REGION Network 2: kontrola przebiegu pętli odczytu parametró z modbus rtu
   RUNG wire#powerrail
      Contact( "dbTags_master_MPP04_2".modbusMaster.busy )
      { S7_Templates := "time_type := Time" } "IEC_Timer_loop_rtu_error_DB".TON(pt := "dbTimersForDrivers".error_loop_modbus_rtu.PT, et =>)
      Coil( "comunication_alarm_modbus_rtu" )
   END_RUNG
   // the same network as SCL:
   "IEC_Timer_loop_rtu_error_DB".TON(IN := "dbTags_master_MPP04_2".modbusMaster.busy,
                           PT := "dbTimersForDrivers".error_loop_modbus_rtu.PT);
   "comunication_alarm_modbus_rtu" := "IEC_Timer_loop_rtu_error_DB".Q;
END_REGION

REGION Network 3: przekazanie do zmiennej error status
   // jeśli wystąpił błąd to przenieś 8200 ( kod brak urządzenia na linni)
   RUNG wire#powerrail
      I_Contact( "FirstScan" )
      Contact( "comunication_alarm_modbus_rtu" )
      Move(in := 33280, out1 => "dbTags_master_MPP04_2".modbusMaster.errorStatus)
   END_RUNG
   // the same network as SCL:
   IF NOT "FirstScan" AND "comunication_alarm_modbus_rtu" THEN
       "dbTags_master_MPP04_2".modbusMaster.errorStatus := 33280;
   END_IF;
END_REGION
END_FUNCTION_BLOCK

ORGANIZATION_BLOCK "Cyclic interrupt"   // OB31, LAD, CyclicInterrupt
{ S7_Optimized_Access := 'TRUE' }
VERSION : 0.1
// stored: AutoNumber true, IsIECCheckEnabled false, SetENOAutomatically false
   VAR_INPUT
      Initial_Call : Bool;   // Initial call of this OB
      Event_Count : Int;   // Events discarded
   END_VAR
   VAR_TEMP
      disconect : Bool;
   END_VAR
BEGIN

REGION Network 1: Reset znacznika automatycznego przekazania wartości na zamykanie
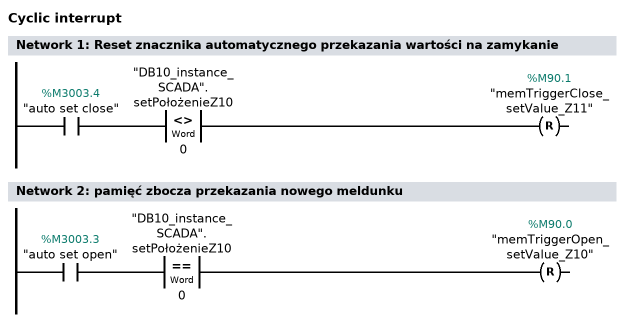
   RUNG wire#powerrail
      Contact( "auto set close" )
      { S7_Templates := "SrcType := Word" } NE_Contact(in1 := "DB10_instance_SCADA".setPołożenieZ10, in2 := 0)
      R_Coil( "memTriggerClose_setValue_Z11" )
   END_RUNG
   // the same network as SCL:
   IF "auto set close" AND ("DB10_instance_SCADA".setPołożenieZ10 <> 0) THEN
       "memTriggerClose_setValue_Z11" := FALSE;
   END_IF;
END_REGION

REGION Network 2: pamięć zbocza przekazania nowego meldunku
   RUNG wire#powerrail
      Contact( "auto set open" )
      { S7_Templates := "SrcType := Word" } EQ_Contact(in1 := "DB10_instance_SCADA".setPołożenieZ10, in2 := 0)
      R_Coil( "memTriggerOpen_setValue_Z10" )
   END_RUNG
   // the same network as SCL:
   IF "auto set open" AND ("DB10_instance_SCADA".setPołożenieZ10 = 0) THEN
       "memTriggerOpen_setValue_Z10" := FALSE;
   END_IF;
END_REGION

REGION Network 3 (SCL): Reset znaczników zbocza wysyłania danych przez TCP
   "memRisingTriger_Data_1" := FALSE;
   "memTrig_Client_Receiving_1" := FALSE;
   "memRisingTriger_Data_2" := FALSE;
   "memTrig_Client_Receiving_2" := FALSE;
   "memRisingTriger_Data_3" := FALSE;
   "memTrig_Client_Receiving_3" := FALSE;
   "memRisingTriger_Data_4" := FALSE;
   "memTrig_Client_Receiving_4" := FALSE;
   "memRisingTriger_Data_5" := FALSE;
   "memTrig_Client_Receiving_5" := FALSE;
   "memRisingTriger_Data_6" := FALSE;
   "memTrig_Client_Receiving_6" := FALSE;
   "memRisingTriger_Data_7" := FALSE;
   "memTrig_Client_Receiving_7" := FALSE;
   "memRisingTriger_Data_8" := FALSE;
   "memTrig_Client_Receiving_8" := FALSE;
   "memRisingTriger_Data_9" := FALSE;
   "memTrig_Client_Receiving_9" := FALSE;
   "memRisingTriger_Data_10" := FALSE;
   "memTrig_Client_Receiving_10" := FALSE;
END_REGION

REGION Network 4 (SCL): pamieć zbocza zmiany danych w zmiennej
   "memRisingTriger_Data_11" := FALSE;
   "memTrig_Client_Receiving_11" := FALSE;
   "memRisingTriger_Data_12" := FALSE;
   "memTrig_Client_Receiving_12" := FALSE;
   "memRisingTriger_Data_13" := FALSE;
   "memTrig_Client_Receiving_13" := FALSE;
   "memRisingTriger_Data_14" := FALSE;
   "memTrig_Client_Receiving_14" := FALSE;
   "memRisingTriger_Data_15" := FALSE;
   "memTrig_Client_Receiving_15" := FALSE;
   "memRisingTriger_Data_16" := FALSE;
   "memTrig_Client_Receiving_16" := FALSE;
   "memRisingTriger_Data_17" := FALSE;
   "memTrig_Client_Receiving_17" := FALSE;
   "memRisingTriger_Data_18" := FALSE;
   "memTrig_Client_Receiving_18" := FALSE;
   "memRisingTriger_Data_19" := FALSE;
   "memTrig_Client_Receiving_19" := FALSE;
   "memRisingTriger_Data_20" := FALSE;
   "memTrig_Client_Receiving_20" := FALSE;
END_REGION

REGION Network 5: pamieć zbocza narastającego przekazania danej do wysłania
END_REGION
END_ORGANIZATION_BLOCK

ORGANIZATION_BLOCK "Cyclic interrupt_ModbusTCP_wysyłanie"   // OB30, LAD, CyclicInterrupt
{ S7_Optimized_Access := 'TRUE' }
VERSION : 0.1
// stored: AutoNumber true, IsIECCheckEnabled false, SetENOAutomatically false
   VAR_INPUT
      Initial_Call : Bool;   // Initial call of this OB
      Event_Count : Int;   // Events discarded
   END_VAR
BEGIN

REGION Network 1: Odczyt poziomów w zbiornku
END_REGION

REGION Network 2 (SCL): Odczyt poziomów w zbiornku
   "AI_poziom_zbiornik_1" := "IW68";
   "AI_poziom_zbiornik_2" := "IW70";
   "AI_poziom_zbiornik_3" := "IW72";
   "AI_poziom_zbiornik_4" := "IW74";

   "AI_położenie_Z10" := "IW78";
END_REGION

REGION Network 3 (SCL): Ciśnienie magistrala

   IF "IW76":P > 0.2 THEN // czy nie uszkodzone rury
     IF "IW76":P < 27651 THEN // przerwana pętla prądowa
       // to przekazanie wartości
       "AI_ciśnienie_B5" := "IW76":P;
       ;
     ELSE
       "AI_ciśnienie_B5" := 32767;
       ;
     END_IF;

     ;
   END_IF;
END_REGION

REGION Network 4 (SCL): Położenie zasuwy Z10
   // Odczyt w FC5
END_REGION
END_ORGANIZATION_BLOCK

ORGANIZATION_BLOCK "Cyclic interrupt_WatchDog_comunication"   // OB32, LAD, CyclicInterrupt
TITLE = Kontrola komunikacji TCP, HMI, PLC
{ S7_Optimized_Access := 'TRUE' }
AUTHOR : rtecmer
VERSION : 0.1
// stored: AutoNumber true, IsIECCheckEnabled false, SetENOAutomatically false
   VAR_INPUT
      Initial_Call : Bool;   // Initial call of this OB
      Event_Count : Int;   // Events discarded
   END_VAR
BEGIN

REGION Network 1
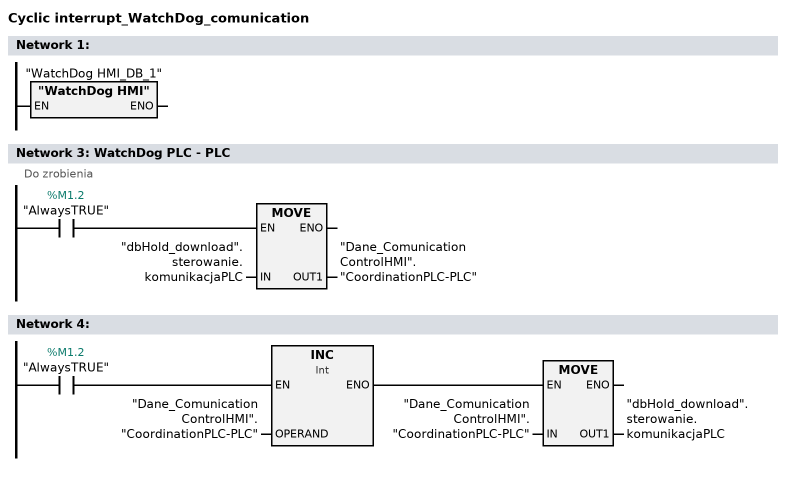
   RUNG wire#powerrail
      "WatchDog HMI_DB_1"()
   END_RUNG
   // the same network as SCL:
   "WatchDog HMI_DB_1"();   // "WatchDog HMI"
END_REGION

REGION Network 3: WatchDog PLC - PLC
   // Do zrobienia
   RUNG wire#powerrail
      Contact( "AlwaysTRUE" )
      Move(in := "dbHold_download".sterowanie.komunikacjaPLC, out1 => "Dane_ComunicationControlHMI"."CoordinationPLC-PLC")
   END_RUNG
   // the same network as SCL:
   IF "AlwaysTRUE" THEN
       "Dane_ComunicationControlHMI"."CoordinationPLC-PLC" := "dbHold_download".sterowanie.komunikacjaPLC;
   END_IF;
END_REGION

REGION Network 4
   RUNG wire#powerrail
      Contact( "AlwaysTRUE" )
      { S7_Templates := "DestType := Int" } Inc( "Dane_ComunicationControlHMI"."CoordinationPLC-PLC" )
      Move(in := "Dane_ComunicationControlHMI"."CoordinationPLC-PLC", out1 => "dbHold_download".sterowanie.komunikacjaPLC)
   END_RUNG
   // the same network as SCL:
   IF "AlwaysTRUE" THEN
       "Dane_ComunicationControlHMI"."CoordinationPLC-PLC" := "Dane_ComunicationControlHMI"."CoordinationPLC-PLC" + 1;
       "dbHold_download".sterowanie.komunikacjaPLC := "Dane_ComunicationControlHMI"."CoordinationPLC-PLC";
   END_IF;
END_REGION

REGION Network 6 (SCL): kasowanie znacznków HMI
   // znaczniki HMI do kasowania alrmów ekranów
   "dbtags_Sterowanie".HMI.resetScreen_1 := FALSE;
   "dbtags_Sterowanie".HMI.resetScreen_2 := FALSE;
   "dbtags_Sterowanie".HMI.resetScreen_3 := FALSE;
   "dbtags_Sterowanie".HMI.resetScreen_4 := FALSE;
   "dbtags_Sterowanie".HMI.resetScreen_5 := FALSE;
   "dbtags_Sterowanie".HMI.resetScreen_6 := FALSE;
   "dbtags_Sterowanie".HMI.resetScreen_7 := FALSE;
   "dbtags_Sterowanie".HMI.resetScreen_8 := FALSE;
END_REGION
END_ORGANIZATION_BLOCK

FUNCTION_BLOCK "WatchDog HMI"   // FB12, LAD
TITLE = WatchDog HMI
{ S7_Optimized_Access := 'TRUE' }
AUTHOR : rtecmer
VERSION : 0.1
// Kontrola komunikacji PLC z HMI. Informacja o zerwanym połączeniu przekazywana do DB SCADA WinCC
// stored: AutoNumber true, IsIECCheckEnabled false, IsRetainMemResEnabled false, MemoryReserve 500, SetENOAutomatically false, UDAEnableTagReadback false
   VAR_TEMP   // added for the SCL form of the ladder/FBD networks
      _w1 : Bool;
      _w2 : Bool;
   END_VAR
BEGIN

REGION Network 1: WatchDog HMI
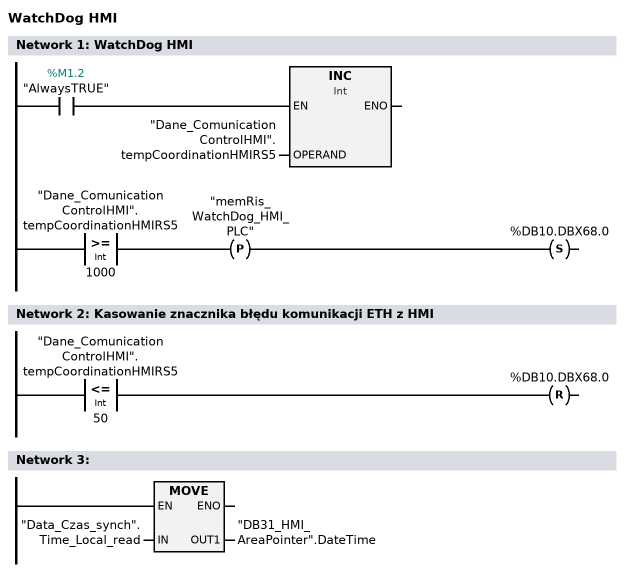
   RUNG wire#powerrail
      Contact( "AlwaysTRUE" )
      { S7_Templates := "DestType := Int" } Inc( "Dane_ComunicationControlHMI".tempCoordinationHMIRS5 )
   END_RUNG
   RUNG wire#powerrail
      { S7_Templates := "SrcType := Int" } GE_Contact(in1 := "Dane_ComunicationControlHMI".tempCoordinationHMIRS5, in2 := 1000)
      P_Trig( "memRis_WatchDog_HMI_PLC" )
      S_Coil( %DB10.DBX68.0 )
   END_RUNG
   // the same network as SCL:
   IF "AlwaysTRUE" THEN
       "Dane_ComunicationControlHMI".tempCoordinationHMIRS5 := "Dane_ComunicationControlHMI".tempCoordinationHMIRS5 + 1;
   END_IF;
   #_w1 := "Dane_ComunicationControlHMI".tempCoordinationHMIRS5 >= 1000;
   #_w2 := #_w1 AND NOT "memRis_WatchDog_HMI_PLC";   // rising edge
   "memRis_WatchDog_HMI_PLC" := #_w1;
   IF #_w2 THEN %DB10.DBX68.0 := TRUE; END_IF;
END_REGION

REGION Network 2: Kasowanie znacznika błędu komunikacji ETH z HMI
   RUNG wire#powerrail
      { S7_Templates := "SrcType := Int" } LE_Contact(in1 := "Dane_ComunicationControlHMI".tempCoordinationHMIRS5, in2 := 50)
      R_Coil( %DB10.DBX68.0 )
   END_RUNG
   // the same network as SCL:
   IF "Dane_ComunicationControlHMI".tempCoordinationHMIRS5 <= 50 THEN %DB10.DBX68.0 := FALSE; END_IF;
END_REGION

REGION Network 3
   RUNG wire#powerrail
      Move(in := "Data_Czas_synch".Time_Local_read, out1 => "DB31_HMI_AreaPointer".DateTime)
   END_RUNG
   // the same network as SCL:
   "DB31_HMI_AreaPointer".DateTime := "Data_Czas_synch".Time_Local_read;
END_REGION
END_FUNCTION_BLOCK

ORGANIZATION_BLOCK "Diagnostic error interrupt"   // OB82, LAD, DiagnosticErrorInterrupt
{ S7_Optimized_Access := 'TRUE' }
VERSION : 0.1
// stored: IsIECCheckEnabled false, SetENOAutomatically false
   VAR_INPUT
      IO_State : Word;   // IO state of the HW object
      LADDR : HW_ANY;   // Hardware identifier
      Channel : UInt;   // Channel number
      MultiError : Bool;   // =true if more than one error is present
   END_VAR
   VAR_TEMP
      RetVal_RD_SYS_T : Int;   // //Status of the instruction RD_SYS_T: Read time-of-day
   END_VAR
BEGIN

REGION Network 2 (SCL)
   "EX012_ErrorBuffer_OB82".OB82ErrorCounter := "EX012_ErrorBuffer_OB82".OB82ErrorCounter + 1;
   //ochrona przed przepełnieniem tabeli
   IF ("EX012_ErrorBuffer_OB82".OB82ErrorCounter > "CONST_BUFFER_OB82") THEN
     "EX012_ErrorBuffer_OB82".OB82ErrorCounter := 1;
   END_IF;
   //Wystąpił błąd czasu
   #RetVal_RD_SYS_T := RD_LOC_T(OUT => "EX012_ErrorBuffer_OB82".ErrorDataOB82["EX012_ErrorBuffer_OB82".OB82ErrorCounter].ErrorTimestamp);
   //Zapis błedu do buffora (ErrorBuffor)
   "EX012_ErrorBuffer_OB82".ErrorDataOB82["EX012_ErrorBuffer_OB82".OB82ErrorCounter].IO_State := #IO_State;
   "EX012_ErrorBuffer_OB82".ErrorDataOB82["EX012_ErrorBuffer_OB82".OB82ErrorCounter].LADDR := #LADDR;
   "EX012_ErrorBuffer_OB82".ErrorDataOB82["EX012_ErrorBuffer_OB82".OB82ErrorCounter].Channel := #Channel;
   "EX012_ErrorBuffer_OB82".ErrorDataOB82["EX012_ErrorBuffer_OB82".OB82ErrorCounter].MultiError := #MultiError;
END_REGION
END_ORGANIZATION_BLOCK

ORGANIZATION_BLOCK "Startup"   // OB100, LAD, Startup
TITLE = "Complete Restart"
{ S7_Optimized_Access := 'TRUE' }
VERSION : 0.1
// Zasuwa status aut. zamknięta= 35980
// Zasuwa status aut. otwarta=34438
// stored: AutoNumber true, IsIECCheckEnabled false, SetENOAutomatically false
   VAR_INPUT
      LostRetentive : Bool;   // True if retentive data are lost
      LostRTC : Bool;   // True if date and time are lost
   END_VAR
BEGIN

REGION Network 1: znacznik powrotu zasilania
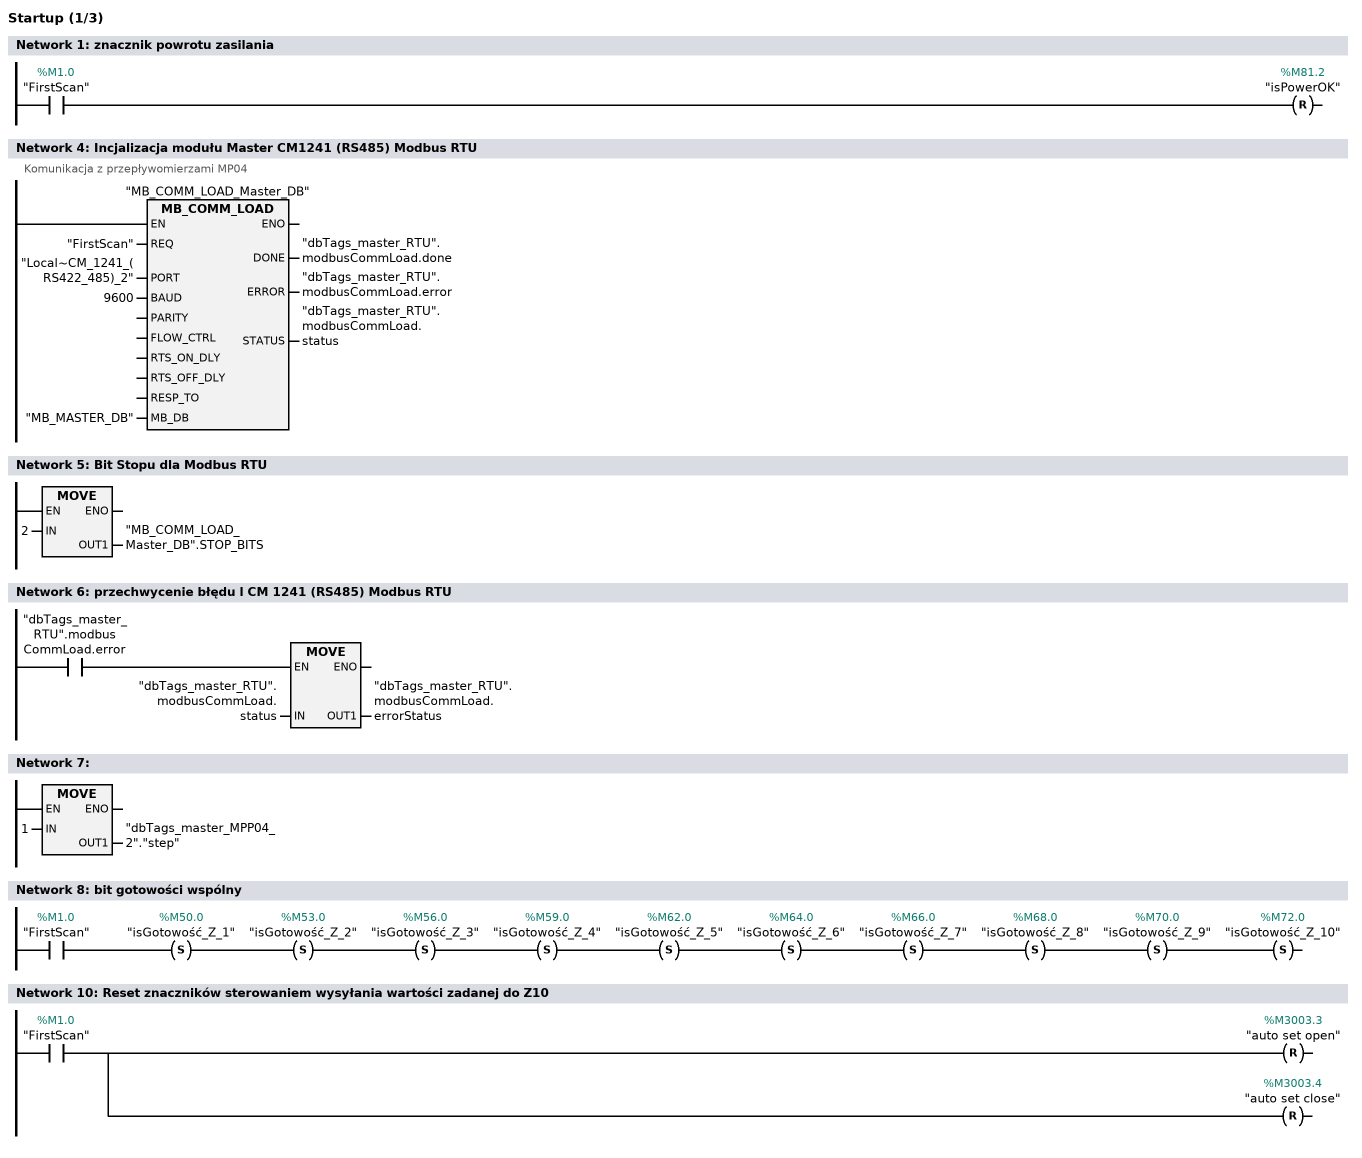
   RUNG wire#powerrail
      Contact( "FirstScan" )
      R_Coil( "isPowerOK" )
   END_RUNG
   // the same network as SCL:
   IF "FirstScan" THEN "isPowerOK" := FALSE; END_IF;
END_REGION

REGION Network 2 (SCL): konfiguracja filtru Kalmana
   IF "FirstScan" THEN //w pierwszym cyklu sterownika
     FOR "I" := 0 TO 3 DO
       "KALMAN_DB".kalman_K["I"] := 0.0;
       "KALMAN_DB".kalman_R["I"] := 0.001;  //niepewność pomiaru
       "KALMAN_DB".kalman_Q["I"] := 0.00001;  //niepewność procesu
       "KALMAN_DB".kalman_P["I"] := 1.0;
     END_FOR;        //parametry R i Q można dobrać osobno dla każdego kanału
   END_IF;           //zostaje wykonana inicjalizacja wszystkich 5 torów analogowych
END_REGION

REGION Network 3 (SCL): Kasowanie alarmów
   "dbtags_Sterowanie".HMI.resetScreen_1 := TRUE;
   "dbtags_Sterowanie".HMI.resetScreen_5 := TRUE;
   "dbtags_Sterowanie".HMI.resetScreen_4 := TRUE;
   "dbtags_Sterowanie".HMI.resetScreen_3 := TRUE;
   "dbtags_Sterowanie".HMI.resetScreen_2 := TRUE;
END_REGION

REGION Network 4: Incjalizacja modułu Master CM1241 (RS485) Modbus RTU
   // Komunikacja z przepływomierzami MP04
   RUNG wire#powerrail
      "MB_COMM_LOAD_Master_DB".MB_COMM_LOAD(REQ := "FirstScan", PORT := "Local~CM_1241_(RS422_485)_2", BAUD := 9600, PARITY :=, FLOW_CTRL :=, RTS_ON_DLY :=, RTS_OFF_DLY :=, RESP_TO :=, MB_DB := "MB_MASTER_DB", DONE => "dbTags_master_RTU".modbusCommLoad.done, ERROR => "dbTags_master_RTU".modbusCommLoad.error, STATUS => "dbTags_master_RTU".modbusCommLoad.status)
   END_RUNG
   // the same network as SCL:
   "MB_COMM_LOAD_Master_DB"(REQ := "FirstScan",   // MB_COMM_LOAD
                           PORT := "Local~CM_1241_(RS422_485)_2",
                           BAUD := 9600,
                           MB_DB := "MB_MASTER_DB",
                           DONE => "dbTags_master_RTU".modbusCommLoad.done,
                           ERROR => "dbTags_master_RTU".modbusCommLoad.error,
                           STATUS => "dbTags_master_RTU".modbusCommLoad.status);
END_REGION

REGION Network 5: Bit Stopu dla Modbus RTU
   RUNG wire#powerrail
      Move(in := 2, out1 => "MB_COMM_LOAD_Master_DB".STOP_BITS)
   END_RUNG
   // the same network as SCL:
   "MB_COMM_LOAD_Master_DB".STOP_BITS := 2;
END_REGION

REGION Network 6: przechwycenie błędu l CM 1241 (RS485) Modbus RTU
   RUNG wire#powerrail
      Contact( "dbTags_master_RTU".modbusCommLoad.error )
      { S7_GenerateENO := "TRUE" } Move(in := "dbTags_master_RTU".modbusCommLoad.status, out1 => "dbTags_master_RTU".modbusCommLoad.errorStatus)
   END_RUNG
   // the same network as SCL:
   IF "dbTags_master_RTU".modbusCommLoad.error THEN
       "dbTags_master_RTU".modbusCommLoad.errorStatus := "dbTags_master_RTU".modbusCommLoad.status;
   END_IF;
END_REGION

REGION Network 7
   RUNG wire#powerrail
      Move(in := 1, out1 => "dbTags_master_MPP04_2"."step")
   END_RUNG
   // the same network as SCL:
   "dbTags_master_MPP04_2"."step" := 1;
END_REGION

REGION Network 8: bit gotowości wspólny
   RUNG wire#powerrail
      Contact( "FirstScan" )
      S_Coil( "isGotowość_Z_1" )
      S_Coil( "isGotowość_Z_2" )
      S_Coil( "isGotowość_Z_3" )
      S_Coil( "isGotowość_Z_4" )
      S_Coil( "isGotowość_Z_5" )
      S_Coil( "isGotowość_Z_6" )
      S_Coil( "isGotowość_Z_7" )
      S_Coil( "isGotowość_Z_8" )
      S_Coil( "isGotowość_Z_9" )
      S_Coil( "isGotowość_Z_10" )
   END_RUNG
   // the same network as SCL:
   IF "FirstScan" THEN
       "isGotowość_Z_1" := TRUE;
       "isGotowość_Z_2" := TRUE;
       "isGotowość_Z_3" := TRUE;
       "isGotowość_Z_4" := TRUE;
       "isGotowość_Z_5" := TRUE;
       "isGotowość_Z_6" := TRUE;
       "isGotowość_Z_7" := TRUE;
       "isGotowość_Z_8" := TRUE;
       "isGotowość_Z_9" := TRUE;
       "isGotowość_Z_10" := TRUE;
   END_IF;
END_REGION

REGION Network 9 (SCL): Wysanie paremetrów sterowania i konfigyracji
     // przekazanie  danych

     "DB10_instance_SCADA".setPołożenieZ10 := "Parametryzacja"."Setting Controll".setPołożenieZ10;
     "DB10_instance_SCADA".ModelSterowania := "Parametryzacja"."Setting Controll".ModelSterowania;
     "DB10_instance_SCADA".TrybSterowania := "Parametryzacja"."Setting Controll".TrybSterowania;
     "DB10_instance_SCADA".setPoziomNapełniania := "Parametryzacja"."Setting Controll".setPoziomNapełniania;
     "DB10_instance_SCADA".setPoziomOpróżnianai := "Parametryzacja"."Setting Controll".setPoziomOpróżnianai;
     // status zasuw
     "DB10_instance_SCADA".instZ1 := "Parametryzacja"."Status drivers".instZ1;
     "DB10_instance_SCADA".instZ2 := "Parametryzacja"."Status drivers".instZ2;
     "DB10_instance_SCADA".instZ3 := "Parametryzacja"."Status drivers".instZ3;
     "DB10_instance_SCADA".instZ4 := "Parametryzacja"."Status drivers".instZ4;
     "DB10_instance_SCADA".instZ5 := "Parametryzacja"."Status drivers".instZ5;
     "DB10_instance_SCADA".instZ6 := "Parametryzacja"."Status drivers".instZ6;
     "DB10_instance_SCADA".instZ7 := "Parametryzacja"."Status drivers".instZ7;
     "DB10_instance_SCADA".instZ8 := "Parametryzacja"."Status drivers".instZ8;
     "DB10_instance_SCADA".instZ9 := "Parametryzacja"."Status drivers".instZ9;
     "DB10_instance_SCADA".instZ10 := "Parametryzacja"."Status drivers".instZ10;

     "DB10_instance_SCADA".actDTL_FillingOn:= "Parametryzacja"."Time Tanks".Start_napełnianie;
     "DB10_instance_SCADA".actDTL_FillingOff:= "Parametryzacja"."Time Tanks".Stop_napełnianie ;
     "DB10_instance_SCADA".actDTL_pumpingOn:= "Parametryzacja"."Time Tanks".Start_przetłaczanie_1 ;
     "DB10_instance_SCADA".actDTL_pumpingOff:= "Parametryzacja"."Time Tanks".Stop_przetłaczanie_1 ;
     "DB10_instance_SCADA".actDTL_RechargingOn:= "Parametryzacja"."Time Tanks".Start_dosilanie_1 ;
     "DB10_instance_SCADA".actDTL_RechargingOff:= "Parametryzacja"."Time Tanks".Stop_dosilanie_1 ;

     "ProcessMemory_Static_1_setChanging" := FALSE;
END_REGION

REGION Network 10: Reset znaczników sterowaniem wysyłania wartości zadanej do Z10
   RUNG wire#powerrail
      Contact( "FirstScan" )
      wire#w1
      R_Coil( "auto set open" )
   END_RUNG
   RUNG wire#w1
      R_Coil( "auto set close" )
   END_RUNG
   // the same network as SCL:
   IF "FirstScan" THEN
       "auto set open" := FALSE;
       "auto set close" := FALSE;
   END_IF;
END_REGION

REGION Network 11: Inicjacja kolejności wywołania Modbus TCP
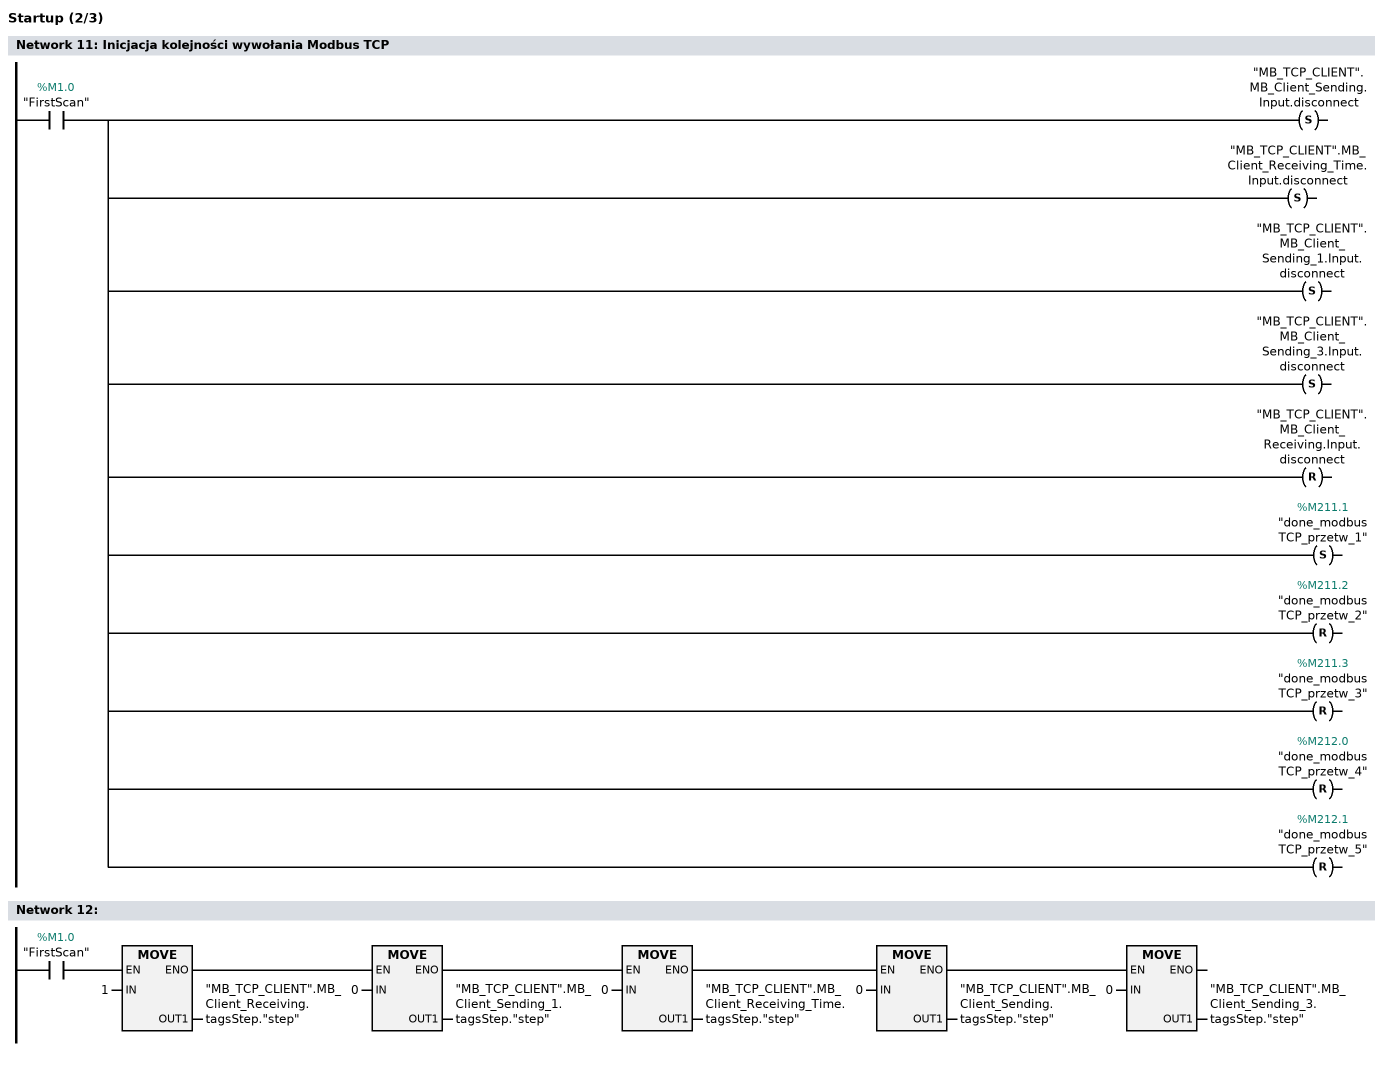
   RUNG wire#powerrail
      Contact( "FirstScan" )
      wire#w1
      S_Coil( "MB_TCP_CLIENT".MB_Client_Sending.Input.disconnect )
   END_RUNG
   RUNG wire#w1
      S_Coil( "MB_TCP_CLIENT".MB_Client_Receiving_Time.Input.disconnect )
   END_RUNG
   RUNG wire#w1
      S_Coil( "MB_TCP_CLIENT".MB_Client_Sending_1.Input.disconnect )
   END_RUNG
   RUNG wire#w1
      S_Coil( "MB_TCP_CLIENT".MB_Client_Sending_3.Input.disconnect )
   END_RUNG
   RUNG wire#w1
      R_Coil( "MB_TCP_CLIENT".MB_Client_Receiving.Input.disconnect )
   END_RUNG
   RUNG wire#w1
      S_Coil( "done_modbusTCP_przetw_1" )
   END_RUNG
   RUNG wire#w1
      R_Coil( "done_modbusTCP_przetw_2" )
   END_RUNG
   RUNG wire#w1
      R_Coil( "done_modbusTCP_przetw_3" )
   END_RUNG
   RUNG wire#w1
      R_Coil( "done_modbusTCP_przetw_4" )
   END_RUNG
   RUNG wire#w1
      R_Coil( "done_modbusTCP_przetw_5" )
   END_RUNG
   // the same network as SCL:
   IF "FirstScan" THEN
       "MB_TCP_CLIENT".MB_Client_Sending.Input.disconnect := TRUE;
       "MB_TCP_CLIENT".MB_Client_Receiving_Time.Input.disconnect := TRUE;
       "MB_TCP_CLIENT".MB_Client_Sending_1.Input.disconnect := TRUE;
       "MB_TCP_CLIENT".MB_Client_Sending_3.Input.disconnect := TRUE;
       "MB_TCP_CLIENT".MB_Client_Receiving.Input.disconnect := FALSE;
       "done_modbusTCP_przetw_1" := TRUE;
       "done_modbusTCP_przetw_2" := FALSE;
       "done_modbusTCP_przetw_3" := FALSE;
       "done_modbusTCP_przetw_4" := FALSE;
       "done_modbusTCP_przetw_5" := FALSE;
   END_IF;
END_REGION

REGION Network 12
   RUNG wire#powerrail
      Contact( "FirstScan" )
      Move(in := 1, out1 => "MB_TCP_CLIENT".MB_Client_Receiving.tagsStep."step")
      Move(in := 0, out1 => "MB_TCP_CLIENT".MB_Client_Sending_1.tagsStep."step")
      Move(in := 0, out1 => "MB_TCP_CLIENT".MB_Client_Receiving_Time.tagsStep."step")
      Move(in := 0, out1 => "MB_TCP_CLIENT".MB_Client_Sending.tagsStep."step")
      Move(in := 0, out1 => "MB_TCP_CLIENT".MB_Client_Sending_3.tagsStep."step")
   END_RUNG
   // the same network as SCL:
   IF "FirstScan" THEN
       "MB_TCP_CLIENT".MB_Client_Receiving.tagsStep."step" := 1;
       "MB_TCP_CLIENT".MB_Client_Sending_1.tagsStep."step" := 0;
       "MB_TCP_CLIENT".MB_Client_Receiving_Time.tagsStep."step" := 0;
       "MB_TCP_CLIENT".MB_Client_Sending.tagsStep."step" := 0;
       "MB_TCP_CLIENT".MB_Client_Sending_3.tagsStep."step" := 0;
   END_IF;
END_REGION

REGION Network 13
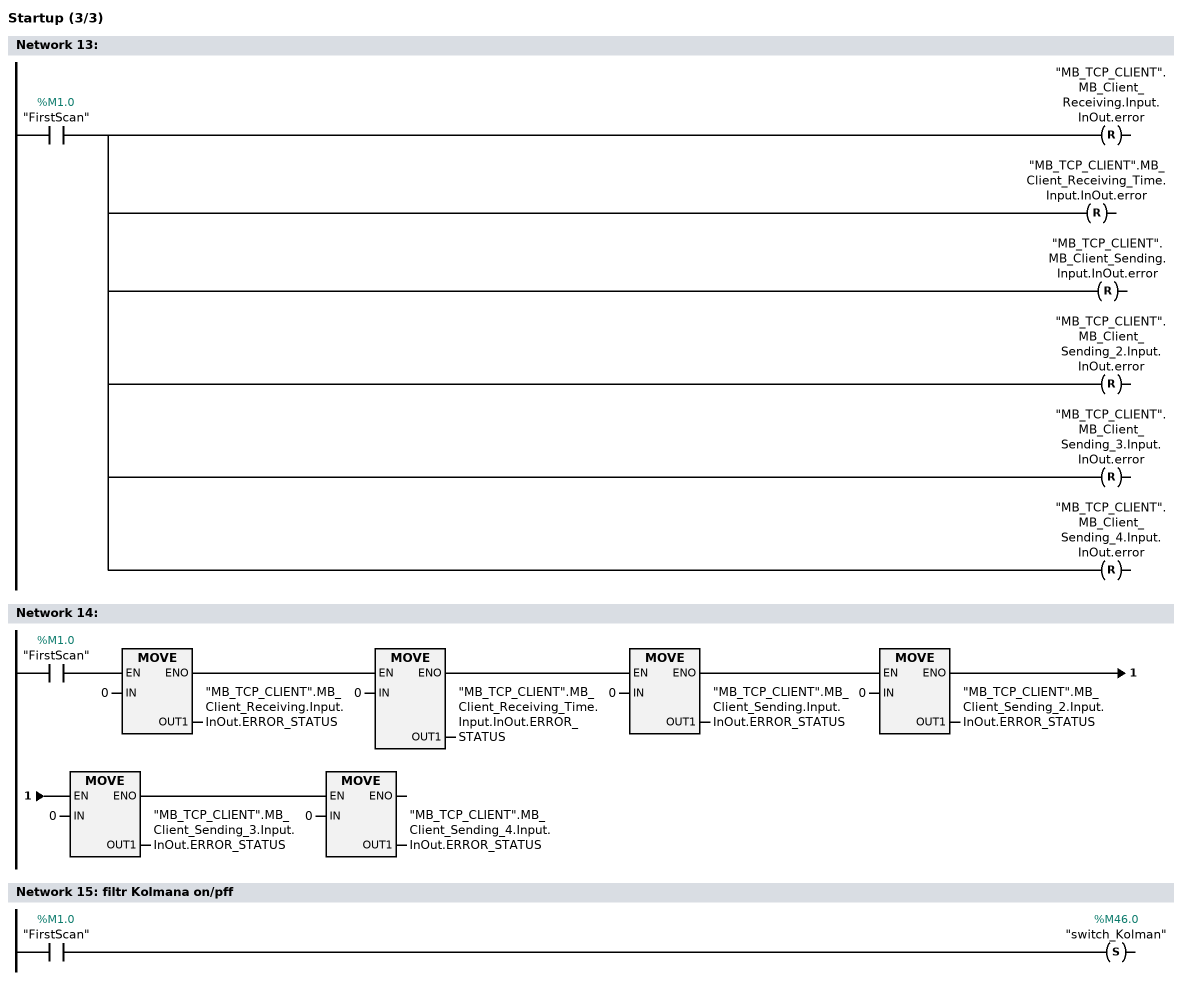
   RUNG wire#powerrail
      Contact( "FirstScan" )
      wire#w1
      R_Coil( "MB_TCP_CLIENT".MB_Client_Receiving.Input.InOut.error )
   END_RUNG
   RUNG wire#w1
      R_Coil( "MB_TCP_CLIENT".MB_Client_Receiving_Time.Input.InOut.error )
   END_RUNG
   RUNG wire#w1
      R_Coil( "MB_TCP_CLIENT".MB_Client_Sending.Input.InOut.error )
   END_RUNG
   RUNG wire#w1
      R_Coil( "MB_TCP_CLIENT".MB_Client_Sending_2.Input.InOut.error )
   END_RUNG
   RUNG wire#w1
      R_Coil( "MB_TCP_CLIENT".MB_Client_Sending_3.Input.InOut.error )
   END_RUNG
   RUNG wire#w1
      R_Coil( "MB_TCP_CLIENT".MB_Client_Sending_4.Input.InOut.error )
   END_RUNG
   // the same network as SCL:
   IF "FirstScan" THEN
       "MB_TCP_CLIENT".MB_Client_Receiving.Input.InOut.error := FALSE;
       "MB_TCP_CLIENT".MB_Client_Receiving_Time.Input.InOut.error := FALSE;
       "MB_TCP_CLIENT".MB_Client_Sending.Input.InOut.error := FALSE;
       "MB_TCP_CLIENT".MB_Client_Sending_2.Input.InOut.error := FALSE;
       "MB_TCP_CLIENT".MB_Client_Sending_3.Input.InOut.error := FALSE;
       "MB_TCP_CLIENT".MB_Client_Sending_4.Input.InOut.error := FALSE;
   END_IF;
END_REGION

REGION Network 14
   RUNG wire#powerrail
      Contact( "FirstScan" )
      Move(in := 0, out1 => "MB_TCP_CLIENT".MB_Client_Receiving.Input.InOut.ERROR_STATUS)
      Move(in := 0, out1 => "MB_TCP_CLIENT".MB_Client_Receiving_Time.Input.InOut.ERROR_STATUS)
      Move(in := 0, out1 => "MB_TCP_CLIENT".MB_Client_Sending.Input.InOut.ERROR_STATUS)
      Move(in := 0, out1 => "MB_TCP_CLIENT".MB_Client_Sending_2.Input.InOut.ERROR_STATUS)
      Move(in := 0, out1 => "MB_TCP_CLIENT".MB_Client_Sending_3.Input.InOut.ERROR_STATUS)
      Move(in := 0, out1 => "MB_TCP_CLIENT".MB_Client_Sending_4.Input.InOut.ERROR_STATUS)
   END_RUNG
   // the same network as SCL:
   IF "FirstScan" THEN
       "MB_TCP_CLIENT".MB_Client_Receiving.Input.InOut.ERROR_STATUS := 0;
       "MB_TCP_CLIENT".MB_Client_Receiving_Time.Input.InOut.ERROR_STATUS := 0;
       "MB_TCP_CLIENT".MB_Client_Sending.Input.InOut.ERROR_STATUS := 0;
       "MB_TCP_CLIENT".MB_Client_Sending_2.Input.InOut.ERROR_STATUS := 0;
       "MB_TCP_CLIENT".MB_Client_Sending_3.Input.InOut.ERROR_STATUS := 0;
       "MB_TCP_CLIENT".MB_Client_Sending_4.Input.InOut.ERROR_STATUS := 0;
   END_IF;
END_REGION

REGION Network 15: filtr Kolmana on/pff
   RUNG wire#powerrail
      Contact( "FirstScan" )
      S_Coil( "switch_Kolman" )
   END_RUNG
   // the same network as SCL:
   IF "FirstScan" THEN "switch_Kolman" := TRUE; END_IF;
END_REGION
END_ORGANIZATION_BLOCK

ORGANIZATION_BLOCK "Time delay interrupt"   // OB20, LAD, TimeDelayInterrupt
{ S7_Optimized_Access := 'TRUE' }
VERSION : 0.1
// stored: AutoNumber true, IsIECCheckEnabled false, SetENOAutomatically false
   VAR_INPUT
      Sign : Word;   // Identifier input (SIGN) passed to triggering call of SRT_DINT
   END_VAR
BEGIN
END_ORGANIZATION_BLOCK

FUNCTION_BLOCK "VLV02_POSITION_old"   // FB17, LAD
TITLE = Valve driver 02
{ S7_Optimized_Access := 'FALSE' }
AUTHOR : RTecmer
VERSION : 0.2
// Driver 0-100% position drives
// Slowo STATUSU Napedu
// STAT - Prawy Byte
// WIZ  - Lewy Byte
//  
//   -STAT wektor stanu zaworu
//     -bit 0- alarm                                  (sygnal do SCADA)
//     -bit 1- zawor otwarty                    (sygnal do SCADA)
//     -bit 2-sterowanie zdal=1 loc=0 (sygnal do SCADA)
//     -bit 3- zawor zamkniety               (sygnal do SCADA)
//     -bit 4-otwieranie reczne              (sygnal z SCADA)
//     -bit 5-zamykanie reczne              (sygnal z SCADA)
//     -bit 6-alarm reset                        (sygnal z SCADA
//     -bit 8-auto= 1man=0                  (sygnal z SCADA)
//   -SUPV 
//   -CLSD zawor zamkniety                    - wejscie
//   -OPND zawor otwarty                        - wejscie
//   -REMT sterowanie zdal=1 loc=0      - wejscie
//   -OPEN otwarcie                                  - wyjscie
//   -CLSE zamkniecie                              - wyjscie
//   - TIM1 czas otwierania  
//   - TIM2 czas zamykania
// stored: AutoNumber false, IsIECCheckEnabled false, SetENOAutomatically false, UDAEnableTagReadback false
   VAR_INPUT
      SetOpen_Percent { ExternalAccessible := 'False'; ExternalVisible := 'False'; ExternalWritable := 'False'} : Word;   // Zadany procent otwarcia
      VectorOut { ExternalAccessible := 'False'; ExternalVisible := 'False'; ExternalWritable := 'False'} : Word;   // Wektor otwarcia z nadajnika
      CLSD : Bool;   // Zamknięta
      OPND : Bool;   // Otwarta
      REMT : Bool;   // Sterowanie zdalne =1, remontowe=0
   END_VAR
   VAR_IN_OUT
      CLSE { ExternalAccessible := 'False'; ExternalVisible := 'False'; ExternalWritable := 'False'} : Bool;   // Wyjście zamykanie
      OPEN { ExternalAccessible := 'False'; ExternalVisible := 'False'; ExternalWritable := 'False'} : Bool;   // Wyjście Otwieranie
      WIZ : Byte;   // Wektor SCADA
      STAT : Byte;   // Wektor statusu napędu
      TMR1 : IEC_TIMER;   // Timer
   END_VAR
   VAR_TEMP
      SVMC : Bool;   // Automat na zamykanie
      SVMO : Bool;   // Automat na otwieranie
      man_Close : Bool;   // znacznik zamykania w trymie manual
      man_Open : Bool;   // znacznik otwierania w trybie manual
      instDiffOpen : Real;   // róznica kąta otwarcia zasuwy
      SP_Real : Real;   // Zadana wartość po konwersji
      PV_Real : Real;   // Vektor położeia po konwerski
      Diff_Real : Real;   // różnica po konwersji
      tmpError_Open : Bool;   // pomocniczy znacznik kontroli czasu jazdy na otwieranie
      tmpError_Close : Bool;   // pomocniczy znacznik kontroli czasu jazdy na zamykanie
   END_VAR
BEGIN

REGION Network 1
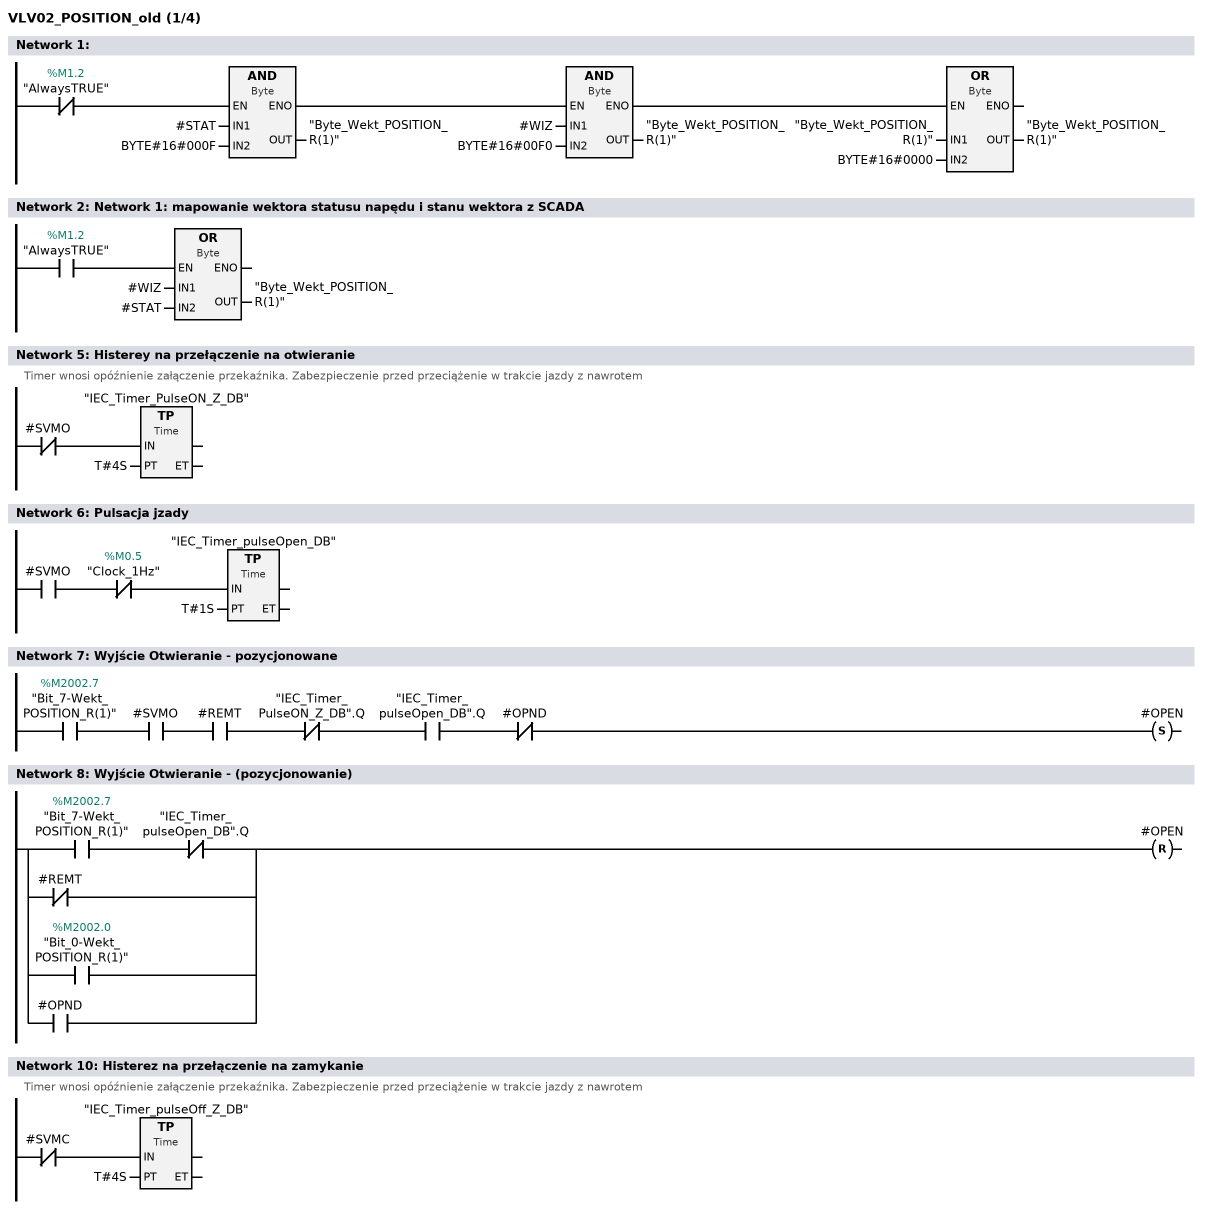
   IF NOT "AlwaysTRUE" THEN
       "Byte_Wekt_POSITION_R(1)" := #STAT AND BYTE#16#000F;
       "Byte_Wekt_POSITION_R(1)" := #WIZ AND BYTE#16#00F0;
       "Byte_Wekt_POSITION_R(1)" := "Byte_Wekt_POSITION_R(1)" OR BYTE#16#0000;
   END_IF;
END_REGION

REGION Network 2: Network 1: mapowanie wektora statusu napędu i stanu wektora z SCADA
   IF "AlwaysTRUE" THEN "Byte_Wekt_POSITION_R(1)" := #WIZ OR #STAT; END_IF;
END_REGION

REGION Network 3 (SCL): wyliczenie różnicy położenia
   //wyliczenie różnicy położenia
   REGION Konwersja zmiennych 
     // Konwersja do Real
     #SP_Real := INT_TO_REAL(#SetOpen_Percent);
     #PV_Real := INT_TO_REAL(#VectorOut);

   END_REGION

   #Diff_Real := (#SP_Real - #PV_Real);
   #instDiffOpen := #Diff_Real;
END_REGION

REGION Network 4 (SCL): Wyznaczenie wektora i jazda na otwierane


   //Strowanie na otwieranie 
   IF #REMT AND ("Bit_0-Wekt_POSITION_R(1)" = FALSE )THEN
     // Porównaj wartość różnicy do 1
     IF #instDiffOpen > 1.0 AND (#OPND = FALSE )AND ("Bit_0-Wekt_POSITION_R(1)" = TRUE) THEN
       // ustaw znacznik automatyczne otwieranie
       #SVMO := TRUE;
       // znacznik do kontroli czasu 
       #tmpError_Open := TRUE;
     ELSE
       #SVMO := FALSE;
       #tmpError_Open:= FALSE
       ;
     END_IF;

     ;
   END_IF;
END_REGION

REGION Network 5: Histerey na przełączenie na otwieranie
   // Timer wnosi opóźnienie załączenie przekaźnika. Zabezpieczenie przed przeciążenie w trakcie jazdy z nawrotem
   RUNG wire#powerrail
      I_Contact( #SVMO )
      { S7_Templates := "time_type := Time" } "IEC_Timer_PulseON_Z_DB".TP(pt := T#4S, et =>)
   END_RUNG
   // the same network as SCL:
   "IEC_Timer_PulseON_Z_DB".TP(IN := NOT #SVMO, PT := T#4S);
END_REGION

REGION Network 6: Pulsacja jzady
   RUNG wire#powerrail
      Contact( #SVMO )
      I_Contact( "Clock_1Hz" )
      { S7_Templates := "time_type := Time" } "IEC_Timer_pulseOpen_DB".TP(pt := T#1S, et =>)
   END_RUNG
   // the same network as SCL:
   "IEC_Timer_pulseOpen_DB".TP(IN := #SVMO AND NOT "Clock_1Hz", PT := T#1S);
END_REGION

REGION Network 7: Wyjście Otwieranie - pozycjonowane
   RUNG wire#powerrail
      Contact( "Bit_7-Wekt_POSITION_R(1)" )
      Contact( #SVMO )
      Contact( #REMT )
      I_Contact( "IEC_Timer_PulseON_Z_DB".Q )
      Contact( "IEC_Timer_pulseOpen_DB".Q )
      I_Contact( #OPND )
      S_Coil( #OPEN )
   END_RUNG
   // the same network as SCL:
   IF "Bit_7-Wekt_POSITION_R(1)" AND #SVMO AND #REMT AND NOT "IEC_Timer_PulseON_Z_DB".Q AND "IEC_Timer_pulseOpen_DB".Q AND NOT #OPND THEN
       #OPEN := TRUE;
   END_IF;
END_REGION

REGION Network 8: Wyjście Otwieranie - (pozycjonowanie)
   RUNG wire#powerrail
      Contact( "Bit_7-Wekt_POSITION_R(1)" )
      I_Contact( "IEC_Timer_pulseOpen_DB".Q )
      wire#w1
      R_Coil( #OPEN )
   END_RUNG
   RUNG wire#powerrail
      I_Contact( #REMT )
   END_RUNG wire#w1
   RUNG wire#powerrail
      Contact( "Bit_0-Wekt_POSITION_R(1)" )
   END_RUNG wire#w1
   RUNG wire#powerrail
      Contact( #OPND )
   END_RUNG wire#w1
   // the same network as SCL:
   IF ("Bit_7-Wekt_POSITION_R(1)" AND NOT "IEC_Timer_pulseOpen_DB".Q) OR NOT #REMT OR "Bit_0-Wekt_POSITION_R(1)" OR #OPND THEN
       #OPEN := FALSE;
   END_IF;
END_REGION

REGION Network 9 (SCL): Wyznaczenie wektora i jazda na zamykanie



   //Strowanie na zamykanie
   IF #REMT AND ("Bit_0-Wekt_POSITION_R(1)" = FALSE )THEN
     // Porównaj wartość różnicy do 1
     IF #instDiffOpen < -1.0 AND (#CLSD = FALSE) AND ("Bit_0-Wekt_POSITION_R(1)" = TRUE) THEN
       // ustaw znacznik automatyczne zamykanie
       #SVMC := TRUE;
       // znacznik kontroli czasu jazdy
       #tmpError_Close := TRUE;
     ELSE
       #SVMC := FALSE;
       #tmpError_Close:= FALSE
       ;
     END_IF;

     ;
   END_IF;
END_REGION

REGION Network 10: Histerez na przełączenie na zamykanie
   // Timer wnosi opóźnienie załączenie przekaźnika. Zabezpieczenie przed przeciążenie w trakcie jazdy z nawrotem
   RUNG wire#powerrail
      I_Contact( #SVMC )
      { S7_Templates := "time_type := Time" } "IEC_Timer_pulseOff_Z_DB".TP(pt := T#4S, et =>)
   END_RUNG
   // the same network as SCL:
   "IEC_Timer_pulseOff_Z_DB".TP(IN := NOT #SVMC, PT := T#4S);
END_REGION

REGION Network 11: Pulsacja jzady
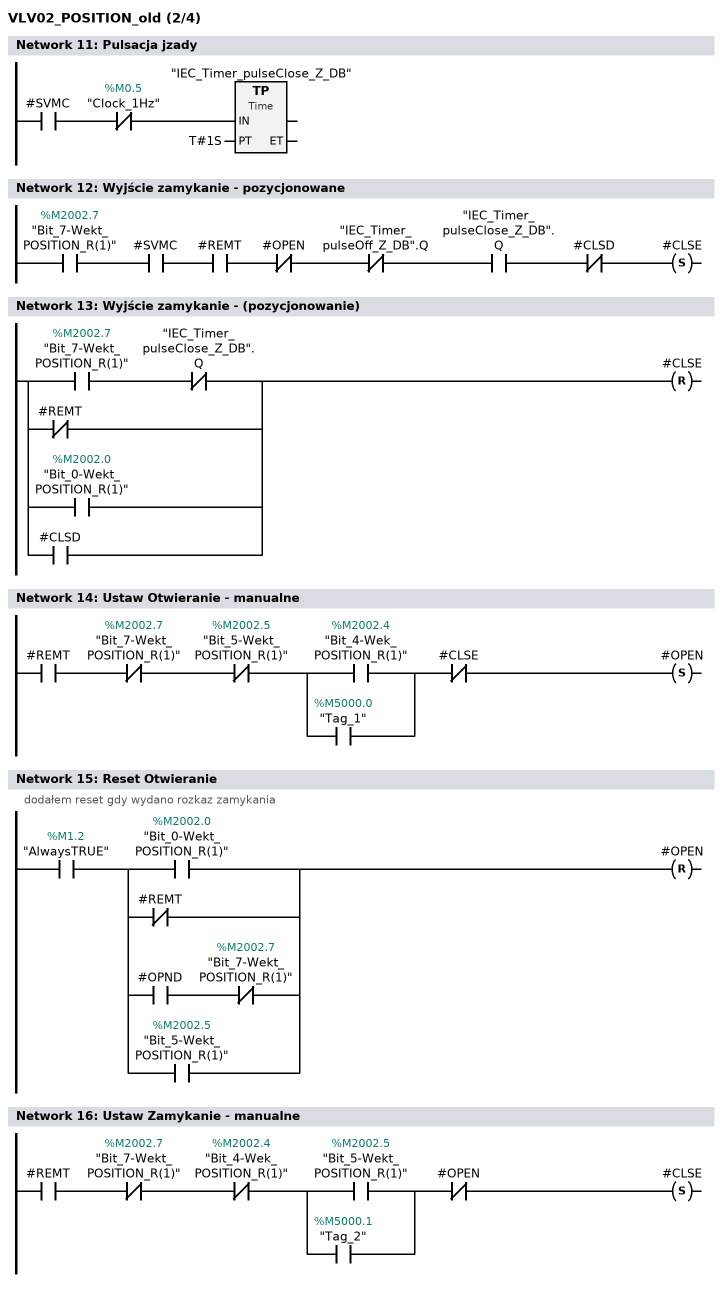
   RUNG wire#powerrail
      Contact( #SVMC )
      I_Contact( "Clock_1Hz" )
      { S7_Templates := "time_type := Time" } "IEC_Timer_pulseClose_Z_DB".TP(pt := T#1S, et =>)
   END_RUNG
   // the same network as SCL:
   "IEC_Timer_pulseClose_Z_DB".TP(IN := #SVMC AND NOT "Clock_1Hz", PT := T#1S);
END_REGION

REGION Network 12: Wyjście zamykanie - pozycjonowane
   RUNG wire#powerrail
      Contact( "Bit_7-Wekt_POSITION_R(1)" )
      Contact( #SVMC )
      Contact( #REMT )
      I_Contact( #OPEN )
      I_Contact( "IEC_Timer_pulseOff_Z_DB".Q )
      Contact( "IEC_Timer_pulseClose_Z_DB".Q )
      I_Contact( #CLSD )
      S_Coil( #CLSE )
   END_RUNG
   // the same network as SCL:
   IF "Bit_7-Wekt_POSITION_R(1)" AND #SVMC AND #REMT AND NOT #OPEN AND NOT "IEC_Timer_pulseOff_Z_DB".Q AND "IEC_Timer_pulseClose_Z_DB".Q AND NOT #CLSD THEN
       #CLSE := TRUE;
   END_IF;
END_REGION

REGION Network 13: Wyjście zamykanie - (pozycjonowanie)
   RUNG wire#powerrail
      Contact( "Bit_7-Wekt_POSITION_R(1)" )
      I_Contact( "IEC_Timer_pulseClose_Z_DB".Q )
      wire#w1
      R_Coil( #CLSE )
   END_RUNG
   RUNG wire#powerrail
      I_Contact( #REMT )
   END_RUNG wire#w1
   RUNG wire#powerrail
      Contact( "Bit_0-Wekt_POSITION_R(1)" )
   END_RUNG wire#w1
   RUNG wire#powerrail
      Contact( #CLSD )
   END_RUNG wire#w1
   // the same network as SCL:
   IF ("Bit_7-Wekt_POSITION_R(1)" AND NOT "IEC_Timer_pulseClose_Z_DB".Q) OR NOT #REMT OR "Bit_0-Wekt_POSITION_R(1)" OR #CLSD THEN
       #CLSE := FALSE;
   END_IF;
END_REGION

REGION Network 14: Ustaw Otwieranie - manualne
   RUNG wire#powerrail
      Contact( #REMT )
      I_Contact( "Bit_7-Wekt_POSITION_R(1)" )
      I_Contact( "Bit_5-Wekt_POSITION_R(1)" )
      wire#w1
      Contact( "Bit_4-Wek_POSITION_R(1)" )
      wire#w2
      I_Contact( #CLSE )
      S_Coil( #OPEN )
   END_RUNG
   RUNG wire#w1
      Contact( "Tag_1" )
   END_RUNG wire#w2
   // the same network as SCL:
   IF #REMT AND NOT "Bit_7-Wekt_POSITION_R(1)" AND NOT "Bit_5-Wekt_POSITION_R(1)" AND ("Bit_4-Wek_POSITION_R(1)" OR "Tag_1") AND NOT #CLSE THEN
       #OPEN := TRUE;
   END_IF;
END_REGION

REGION Network 15: Reset Otwieranie
   // dodałem reset gdy wydano rozkaz zamykania
   RUNG wire#powerrail
      Contact( "AlwaysTRUE" )
      wire#w1
      Contact( "Bit_0-Wekt_POSITION_R(1)" )
      wire#w2
      R_Coil( #OPEN )
   END_RUNG
   RUNG wire#w1
      I_Contact( #REMT )
   END_RUNG wire#w2
   RUNG wire#w1
      Contact( #OPND )
      I_Contact( "Bit_7-Wekt_POSITION_R(1)" )
   END_RUNG wire#w2
   RUNG wire#w1
      Contact( "Bit_5-Wekt_POSITION_R(1)" )
   END_RUNG wire#w2
   // the same network as SCL:
   IF "AlwaysTRUE" AND ("Bit_0-Wekt_POSITION_R(1)" OR NOT #REMT OR (#OPND AND NOT "Bit_7-Wekt_POSITION_R(1)") OR "Bit_5-Wekt_POSITION_R(1)") THEN
       #OPEN := FALSE;
   END_IF;
END_REGION

REGION Network 16: Ustaw Zamykanie - manualne
   RUNG wire#powerrail
      Contact( #REMT )
      I_Contact( "Bit_7-Wekt_POSITION_R(1)" )
      I_Contact( "Bit_4-Wek_POSITION_R(1)" )
      wire#w1
      Contact( "Bit_5-Wekt_POSITION_R(1)" )
      wire#w2
      I_Contact( #OPEN )
      S_Coil( #CLSE )
   END_RUNG
   RUNG wire#w1
      Contact( "Tag_2" )
   END_RUNG wire#w2
   // the same network as SCL:
   IF #REMT AND NOT "Bit_7-Wekt_POSITION_R(1)" AND NOT "Bit_4-Wek_POSITION_R(1)" AND ("Bit_5-Wekt_POSITION_R(1)" OR "Tag_2") AND NOT #OPEN THEN
       #CLSE := TRUE;
   END_IF;
END_REGION

REGION Network 17: Reset Zamykanie
   // dodałem reset gdy wydano rozkaz otwierania
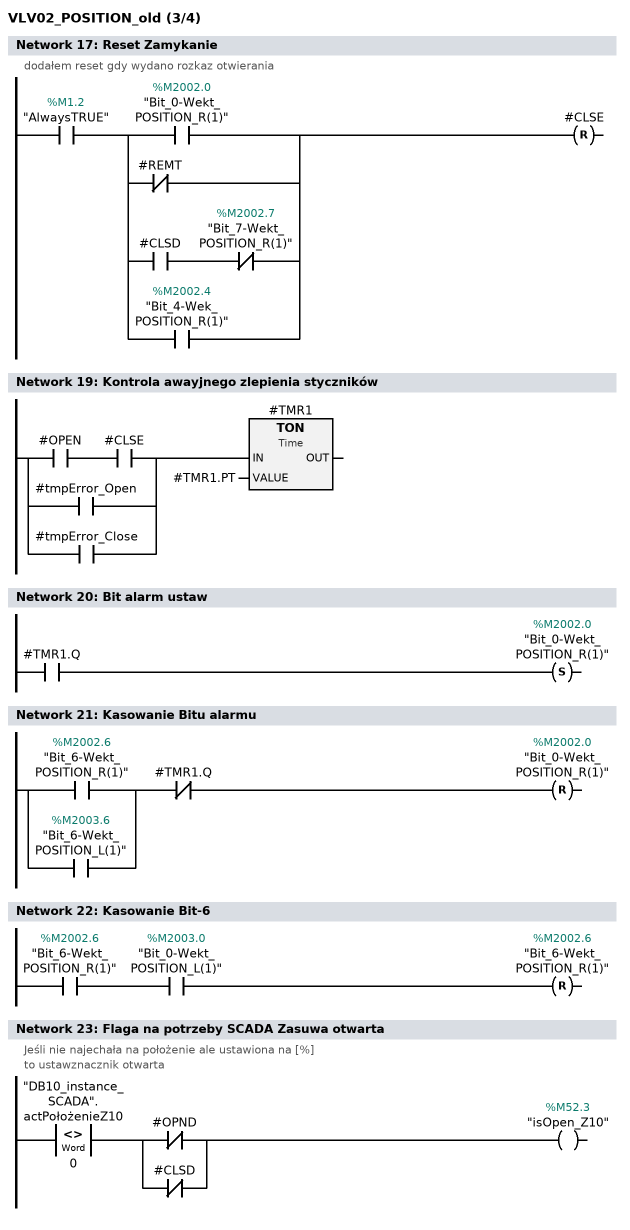
   RUNG wire#powerrail
      Contact( "AlwaysTRUE" )
      wire#w1
      Contact( "Bit_0-Wekt_POSITION_R(1)" )
      wire#w2
      R_Coil( #CLSE )
   END_RUNG
   RUNG wire#w1
      I_Contact( #REMT )
   END_RUNG wire#w2
   RUNG wire#w1
      Contact( #CLSD )
      I_Contact( "Bit_7-Wekt_POSITION_R(1)" )
   END_RUNG wire#w2
   RUNG wire#w1
      Contact( "Bit_4-Wek_POSITION_R(1)" )
   END_RUNG wire#w2
   // the same network as SCL:
   IF "AlwaysTRUE" AND ("Bit_0-Wekt_POSITION_R(1)" OR NOT #REMT OR (#CLSD AND NOT "Bit_7-Wekt_POSITION_R(1)") OR "Bit_4-Wek_POSITION_R(1)") THEN
       #CLSE := FALSE;
   END_IF;
END_REGION

REGION Network 19: Kontrola awayjnego zlepienia styczników
   #TMR1.TON(IN := (#OPEN AND #CLSE) OR #tmpError_Open OR #tmpError_Close, PT := #TMR1.PT);   // TON coil
END_REGION

REGION Network 20: Bit alarm ustaw
   RUNG wire#powerrail
      Contact( #TMR1.Q )
      S_Coil( "Bit_0-Wekt_POSITION_R(1)" )
   END_RUNG
   // the same network as SCL:
   IF #TMR1.Q THEN "Bit_0-Wekt_POSITION_R(1)" := TRUE; END_IF;
END_REGION

REGION Network 21: Kasowanie Bitu alarmu
   RUNG wire#powerrail
      Contact( "Bit_6-Wekt_POSITION_R(1)" )
      wire#w1
      I_Contact( #TMR1.Q )
      R_Coil( "Bit_0-Wekt_POSITION_R(1)" )
   END_RUNG
   RUNG wire#powerrail
      Contact( "Bit_6-Wekt_POSITION_L(1)" )
   END_RUNG wire#w1
   // the same network as SCL:
   IF ("Bit_6-Wekt_POSITION_R(1)" OR "Bit_6-Wekt_POSITION_L(1)") AND NOT #TMR1.Q THEN
       "Bit_0-Wekt_POSITION_R(1)" := FALSE;
   END_IF;
END_REGION

REGION Network 22: Kasowanie Bit-6
   RUNG wire#powerrail
      Contact( "Bit_6-Wekt_POSITION_R(1)" )
      Contact( "Bit_0-Wekt_POSITION_L(1)" )
      R_Coil( "Bit_6-Wekt_POSITION_R(1)" )
   END_RUNG
   // the same network as SCL:
   IF "Bit_6-Wekt_POSITION_R(1)" AND "Bit_0-Wekt_POSITION_L(1)" THEN
       "Bit_6-Wekt_POSITION_R(1)" := FALSE;
   END_IF;
END_REGION

REGION Network 23: Flaga na potrzeby SCADA Zasuwa otwarta
   // Jeśli nie najechała na położenie ale ustawiona na [%]
   // to ustawznacznik otwarta
   RUNG wire#powerrail
      { S7_Templates := "SrcType := Word" } NE_Contact(in1 := "DB10_instance_SCADA".actPołożenieZ10, in2 := 0)
      wire#w1
      I_Contact( #OPND )
      wire#w2
      Coil( "isOpen_Z10" )
   END_RUNG
   RUNG wire#w1
      I_Contact( #CLSD )
   END_RUNG wire#w2
   // the same network as SCL:
   "isOpen_Z10" := ("DB10_instance_SCADA".actPołożenieZ10 <> 0) AND (NOT #OPND OR NOT #CLSD);
END_REGION

REGION Network 24: Przepisanie Byte Wektora napędu
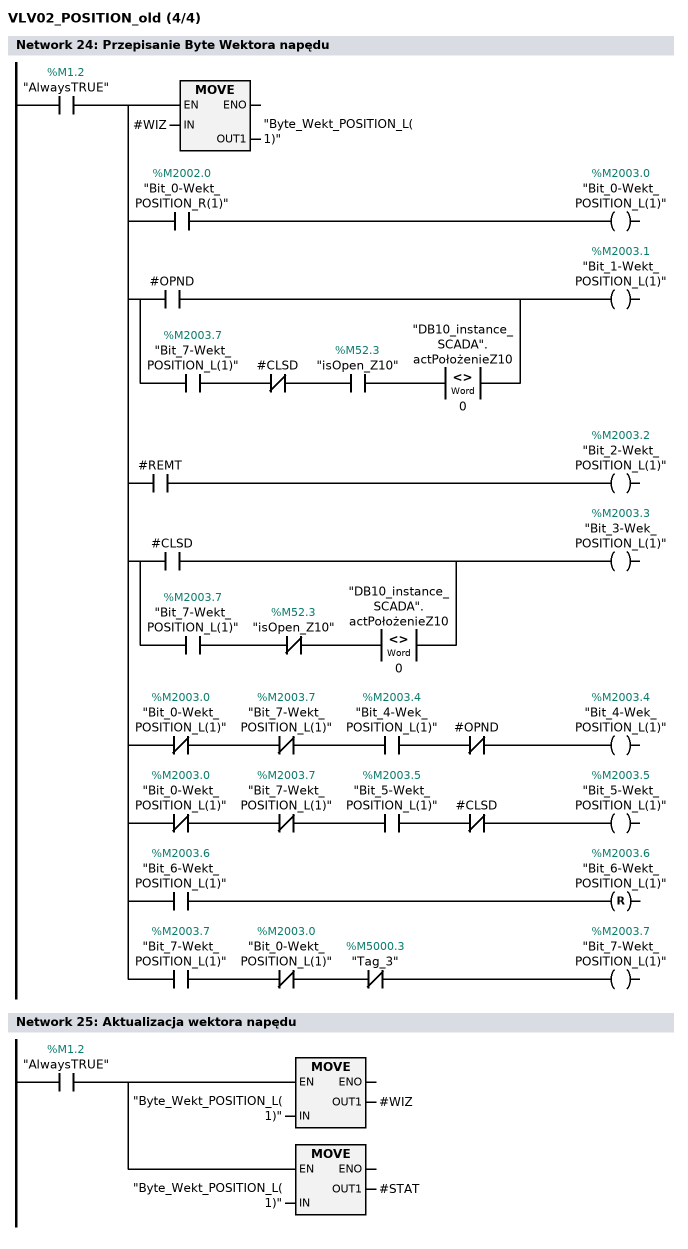
   RUNG wire#powerrail
      Contact( "AlwaysTRUE" )
      wire#w1
      { S7_GenerateENO := "TRUE" } Move(in := #WIZ, out1 => "Byte_Wekt_POSITION_L(1)")
   END_RUNG
   RUNG wire#w1
      Contact( "Bit_0-Wekt_POSITION_R(1)" )
      Coil( "Bit_0-Wekt_POSITION_L(1)" )
   END_RUNG
   RUNG wire#w1
      Contact( #OPND )
      wire#w2
      Coil( "Bit_1-Wekt_POSITION_L(1)" )
   END_RUNG
   RUNG wire#w1
      Contact( "Bit_7-Wekt_POSITION_L(1)" )
      I_Contact( #CLSD )
      Contact( "isOpen_Z10" )
      { S7_Templates := "SrcType := Word" } NE_Contact(in1 := "DB10_instance_SCADA".actPołożenieZ10, in2 := 0)
   END_RUNG wire#w2
   RUNG wire#w1
      Contact( #REMT )
      Coil( "Bit_2-Wekt_POSITION_L(1)" )
   END_RUNG
   RUNG wire#w1
      Contact( #CLSD )
      wire#w3
      Coil( "Bit_3-Wek_POSITION_L(1)" )
   END_RUNG
   RUNG wire#w1
      Contact( "Bit_7-Wekt_POSITION_L(1)" )
      I_Contact( "isOpen_Z10" )
      { S7_Templates := "SrcType := Word" } NE_Contact(in1 := "DB10_instance_SCADA".actPołożenieZ10, in2 := 0)
   END_RUNG wire#w3
   RUNG wire#w1
      I_Contact( "Bit_0-Wekt_POSITION_L(1)" )
      I_Contact( "Bit_7-Wekt_POSITION_L(1)" )
      Contact( "Bit_4-Wek_POSITION_L(1)" )
      I_Contact( #OPND )
      Coil( "Bit_4-Wek_POSITION_L(1)" )
   END_RUNG
   RUNG wire#w1
      I_Contact( "Bit_0-Wekt_POSITION_L(1)" )
      I_Contact( "Bit_7-Wekt_POSITION_L(1)" )
      Contact( "Bit_5-Wekt_POSITION_L(1)" )
      I_Contact( #CLSD )
      Coil( "Bit_5-Wekt_POSITION_L(1)" )
   END_RUNG
   RUNG wire#w1
      Contact( "Bit_6-Wekt_POSITION_L(1)" )
      R_Coil( "Bit_6-Wekt_POSITION_L(1)" )
   END_RUNG
   RUNG wire#w1
      Contact( "Bit_7-Wekt_POSITION_L(1)" )
      I_Contact( "Bit_0-Wekt_POSITION_L(1)" )
      I_Contact( "Tag_3" )
      Coil( "Bit_7-Wekt_POSITION_L(1)" )
   END_RUNG
   // the same network as SCL:
   IF "AlwaysTRUE" THEN "Byte_Wekt_POSITION_L(1)" := #WIZ; END_IF;
   "Bit_0-Wekt_POSITION_L(1)" := "AlwaysTRUE" AND "Bit_0-Wekt_POSITION_R(1)";
   "Bit_1-Wekt_POSITION_L(1)" := "AlwaysTRUE" AND (#OPND OR ("Bit_7-Wekt_POSITION_L(1)" AND NOT #CLSD AND "isOpen_Z10" AND ("DB10_instance_SCADA".actPołożenieZ10 <> 0)));
   "Bit_2-Wekt_POSITION_L(1)" := "AlwaysTRUE" AND #REMT;
   "Bit_3-Wek_POSITION_L(1)" := "AlwaysTRUE" AND (#CLSD OR ("Bit_7-Wekt_POSITION_L(1)" AND NOT "isOpen_Z10" AND ("DB10_instance_SCADA".actPołożenieZ10 <> 0)));
   "Bit_4-Wek_POSITION_L(1)" := "AlwaysTRUE" AND NOT "Bit_0-Wekt_POSITION_L(1)" AND NOT "Bit_7-Wekt_POSITION_L(1)" AND "Bit_4-Wek_POSITION_L(1)" AND NOT #OPND;
   "Bit_5-Wekt_POSITION_L(1)" := "AlwaysTRUE" AND NOT "Bit_0-Wekt_POSITION_L(1)" AND NOT "Bit_7-Wekt_POSITION_L(1)" AND "Bit_5-Wekt_POSITION_L(1)" AND NOT #CLSD;
   IF "AlwaysTRUE" AND "Bit_6-Wekt_POSITION_L(1)" THEN "Bit_6-Wekt_POSITION_L(1)" := FALSE; END_IF;
   "Bit_7-Wekt_POSITION_L(1)" := "AlwaysTRUE" AND "Bit_7-Wekt_POSITION_L(1)" AND NOT "Bit_0-Wekt_POSITION_L(1)" AND NOT "Tag_3";
END_REGION

REGION Network 25: Aktualizacja wektora napędu
   RUNG wire#powerrail
      Contact( "AlwaysTRUE" )
      wire#w1
      { S7_GenerateENO := "TRUE" } Move(in := "Byte_Wekt_POSITION_L(1)", out1 => #WIZ)
   END_RUNG
   RUNG wire#w1
      { S7_GenerateENO := "TRUE" } Move(in := "Byte_Wekt_POSITION_L(1)", out1 => #STAT)
   END_RUNG
   // the same network as SCL:
   IF "AlwaysTRUE" THEN
       #WIZ := "Byte_Wekt_POSITION_L(1)";
       #STAT := "Byte_Wekt_POSITION_L(1)";
   END_IF;
END_REGION
END_FUNCTION_BLOCK

FUNCTION_BLOCK "generator_weekday"   // FB10, LAD
{ S7_Optimized_Access := 'TRUE' }
AUTHOR : RTecmer
FAMILY : XMHour
VERSION : 0.1
// Licznik czasu pracy
// stored: AutoNumber false, IsIECCheckEnabled false, IsRetainMemResEnabled false, MemoryReserve 500, SetENOAutomatically false, UDAEnableTagReadback false
   VAR_INPUT
      Reset { ExternalAccessible := 'False'; ExternalVisible := 'False'; ExternalWritable := 'False'} : Bool;
      Run_WEEKDAY : Bool;
   END_VAR
   VAR_OUTPUT
      Out_Weekday : Bool;   // znacznik
   END_VAR
   VAR_IN_OUT
      Data_sek : Int;
      Data_hour : DWord;
      Edge_Hz { ExternalAccessible := 'False'; ExternalVisible := 'False'; ExternalWritable := 'False'} : Bool;
   END_VAR
   VAR
      sek_real { ExternalAccessible := 'False'; ExternalVisible := 'False'; ExternalWritable := 'False'} : Real;   // pomocnicza konwerski sekund
      hour_sek { ExternalAccessible := 'False'; ExternalVisible := 'False'; ExternalWritable := 'False'} : Real;
      memTrig_Week : Bool;   // pamieć zbocza uruchomienia funkcji tygodniowej
      start_weekday : Bool;   // aktywacja funkcji w cyklu tygodniowym
      tmp_weekend : USInt;   // przechwycona liczba tygodni podczas startu funkcji
   END_VAR
   VAR_TEMP   // added for the SCL form of the ladder/FBD networks
      _w1 : Bool;
      _w2 : Bool;
   END_VAR
BEGIN

REGION Network 1
   // reset liczników po dobie pracy w cyklu tygodniowym
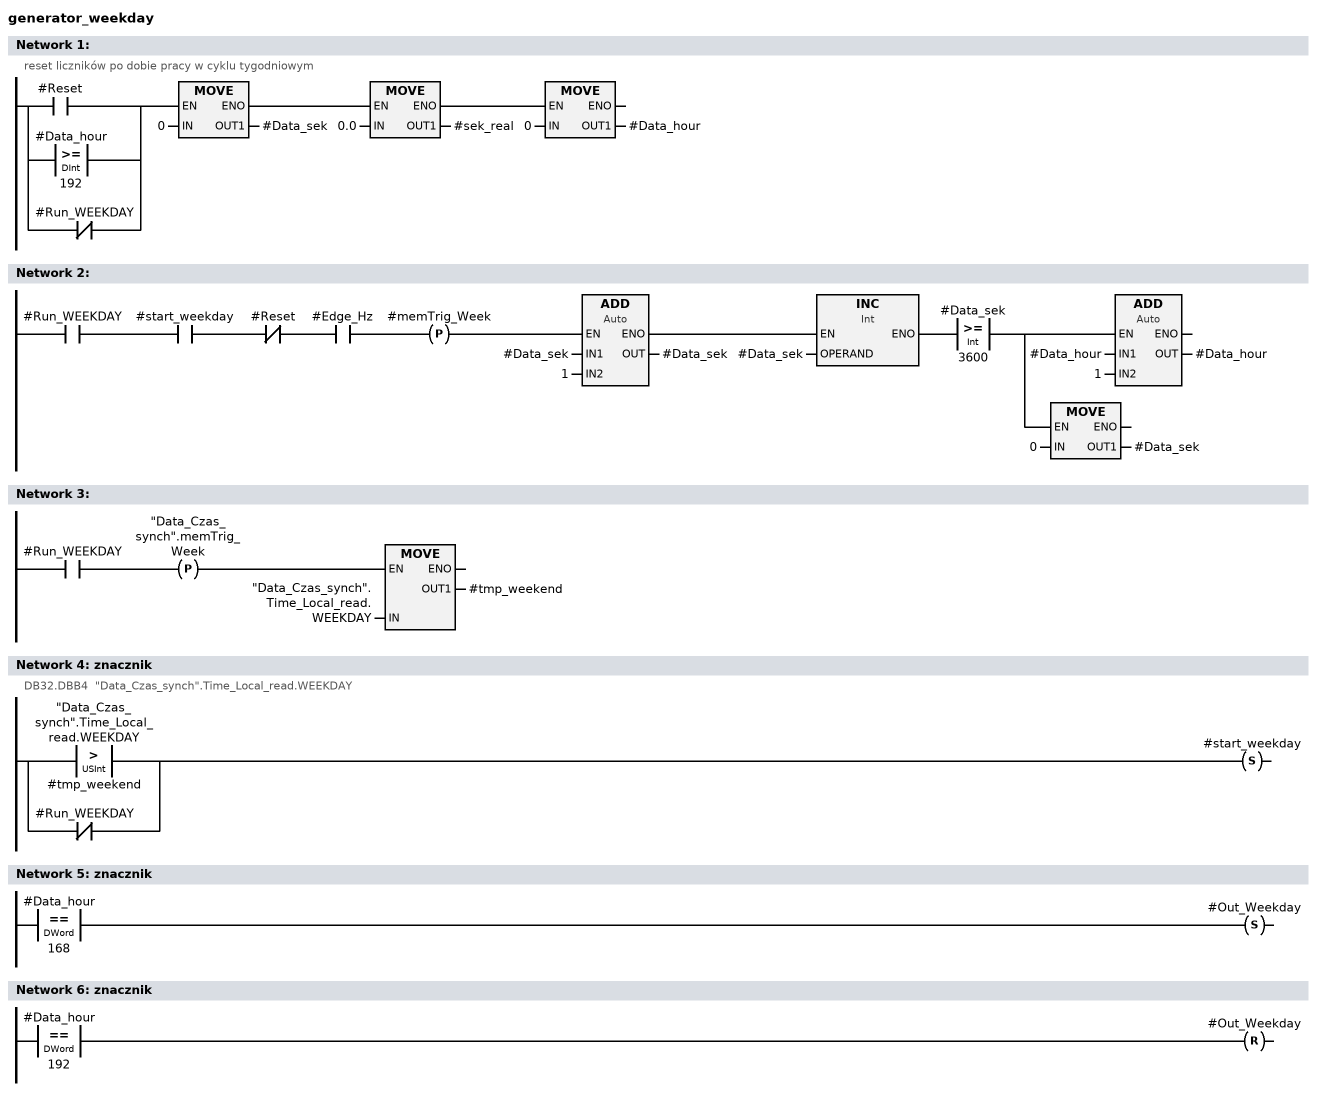
   RUNG wire#powerrail
      Contact( #Reset )
      wire#w1
      { S7_GenerateENO := "TRUE" } Move(in := 0, out1 => #Data_sek)
      { S7_GenerateENO := "TRUE" } Move(in := 0.0, out1 => #sek_real)
      { S7_GenerateENO := "TRUE" } Move(in := 0, out1 => #Data_hour)
   END_RUNG
   RUNG wire#powerrail
      { S7_Templates := "SrcType := DInt" } GE_Contact(in1 := #Data_hour, in2 := 192)
   END_RUNG wire#w1
   RUNG wire#powerrail
      I_Contact( #Run_WEEKDAY )
   END_RUNG wire#w1
   // the same network as SCL:
   // ENO of a box is taken as its EN; it also drops when the box reports an error
   IF #Reset OR (#Data_hour >= 192) OR NOT #Run_WEEKDAY THEN
       #Data_sek := 0;
       #sek_real := 0.0;
       #Data_hour := 0;
   END_IF;
END_REGION

REGION Network 2
   RUNG wire#powerrail
      Contact( #Run_WEEKDAY )
      Contact( #start_weekday )
      I_Contact( #Reset )
      Contact( #Edge_Hz )
      P_Trig( #memTrig_Week )
      { S7_GenerateENO := "TRUE" } Add(in1 := #Data_sek, in2 := 1, out => #Data_sek)
      { S7_Templates := "DestType := Int"; S7_GenerateENO := "TRUE" } Inc( #Data_sek )
      { S7_Templates := "SrcType := Int" } GE_Contact(in1 := #Data_sek, in2 := 3600)
      wire#w1
      { S7_GenerateENO := "TRUE" } Add(in1 := #Data_hour, in2 := 1, out => #Data_hour)
   END_RUNG
   RUNG wire#w1
      { S7_GenerateENO := "TRUE" } Move(in := 0, out1 => #Data_sek)
   END_RUNG
   // the same network as SCL:
   // ENO of a box is taken as its EN; it also drops when the box reports an error
   #_w1 := #Run_WEEKDAY AND #start_weekday AND NOT #Reset AND #Edge_Hz;
   #_w2 := #_w1 AND NOT #memTrig_Week;   // rising edge
   #memTrig_Week := #_w1;
   IF #_w2 THEN
       #Data_sek := #Data_sek + 1;
       #Data_sek := #Data_sek + 1;
   END_IF;
   IF #_w2 AND (#Data_sek >= 3600) THEN
       #Data_hour := #Data_hour + 1;
       #Data_sek := 0;
   END_IF;
END_REGION

REGION Network 3
   RUNG wire#powerrail
      Contact( #Run_WEEKDAY )
      P_Trig( "Data_Czas_synch".memTrig_Week )
      Move(in := "Data_Czas_synch".Time_Local_read.WEEKDAY, out1 => #tmp_weekend)
   END_RUNG
   // the same network as SCL:
   #_w1 := #Run_WEEKDAY AND NOT "Data_Czas_synch".memTrig_Week;   // rising edge
   "Data_Czas_synch".memTrig_Week := #Run_WEEKDAY;
   IF #_w1 THEN #tmp_weekend := "Data_Czas_synch".Time_Local_read.WEEKDAY; END_IF;
END_REGION

REGION Network 4: znacznik
   // DB32.DBB4  "Data_Czas_synch".Time_Local_read.WEEKDAY
   RUNG wire#powerrail
      { S7_Templates := "SrcType := USInt" } GT_Contact(in1 := "Data_Czas_synch".Time_Local_read.WEEKDAY, in2 := #tmp_weekend)
      wire#w1
      S_Coil( #start_weekday )
   END_RUNG
   RUNG wire#powerrail
      I_Contact( #Run_WEEKDAY )
   END_RUNG wire#w1
   // the same network as SCL:
   IF ("Data_Czas_synch".Time_Local_read.WEEKDAY > #tmp_weekend) OR NOT #Run_WEEKDAY THEN
       #start_weekday := TRUE;
   END_IF;
END_REGION

REGION Network 5: znacznik
   RUNG wire#powerrail
      { S7_Templates := "SrcType := DWord" } EQ_Contact(in1 := #Data_hour, in2 := 168)
      S_Coil( #Out_Weekday )
   END_RUNG
   // the same network as SCL:
   IF #Data_hour = 168 THEN #Out_Weekday := TRUE; END_IF;
END_REGION

REGION Network 6: znacznik
   RUNG wire#powerrail
      { S7_Templates := "SrcType := DWord" } EQ_Contact(in1 := #Data_hour, in2 := 192)
      R_Coil( #Out_Weekday )
   END_RUNG
   // the same network as SCL:
   IF #Data_hour = 192 THEN #Out_Weekday := FALSE; END_IF;
END_REGION
END_FUNCTION_BLOCK

FUNCTION "Gotowość_Napędów" : Void   // FC23, LAD
TITLE = Ustawienie Gotowośći
{ S7_Optimized_Access := 'TRUE' }
AUTHOR : rtecmer
VERSION : 0.1
// Funkcja w zależności od przełącznika technologiczne związanego z przebudową zasuw z Czeskich na AUMA przełącza sygnał godowości w zależności jak ajest zasuwa podłączona w procesie technologicznym
// stored: AutoNumber true, IsIECCheckEnabled false, SetENOAutomatically false, UDAEnableTagReadback false
   VAR_TEMP   // added for the SCL form of the ladder/FBD networks
      _w1 : Bool;
   END_VAR
BEGIN

REGION Network 2: bit gotowości wspólny Z1
   // AUMA
   // MODACT MOK250
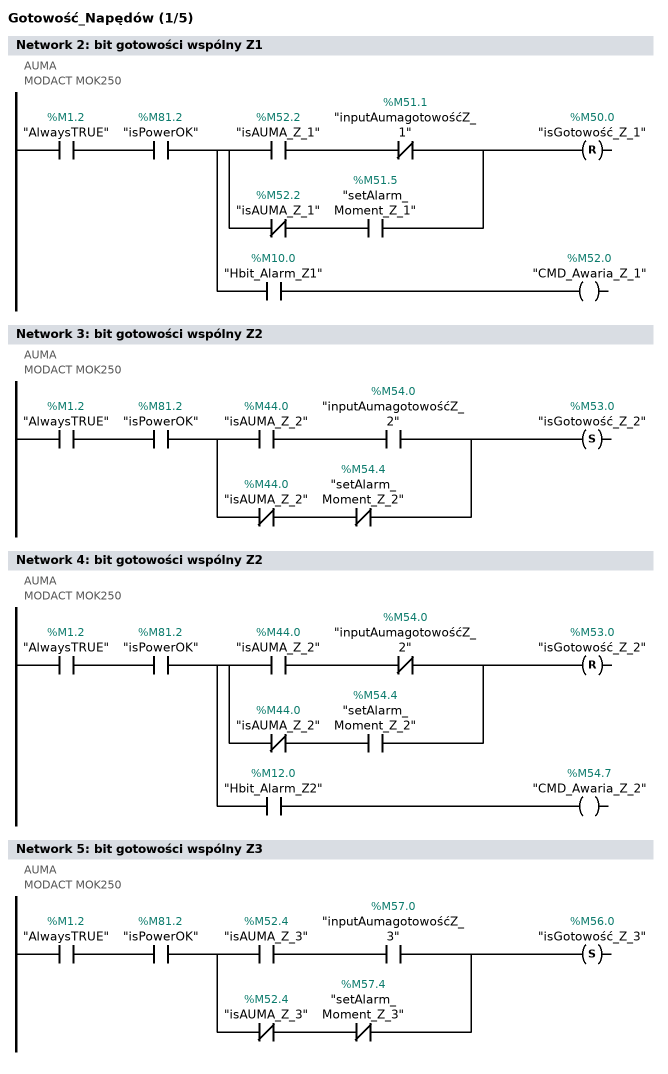
   RUNG wire#powerrail
      Contact( "AlwaysTRUE" )
      Contact( "isPowerOK" )
      wire#w1
      Contact( "isAUMA_Z_1" )
      I_Contact( "inputAumagotowośćZ_1" )
      wire#w2
      R_Coil( "isGotowość_Z_1" )
   END_RUNG
   RUNG wire#w1
      I_Contact( "isAUMA_Z_1" )
      Contact( "setAlarm_Moment_Z_1" )
   END_RUNG wire#w2
   RUNG wire#w1
      Contact( "Hbit_Alarm_Z1" )
      Coil( "CMD_Awaria_Z_1" )
   END_RUNG
   // the same network as SCL:
   #_w1 := "AlwaysTRUE" AND "isPowerOK";
   IF #_w1 AND (("isAUMA_Z_1" AND NOT "inputAumagotowośćZ_1") OR (NOT "isAUMA_Z_1" AND "setAlarm_Moment_Z_1")) THEN
       "isGotowość_Z_1" := FALSE;
   END_IF;
   "CMD_Awaria_Z_1" := #_w1 AND "Hbit_Alarm_Z1";
END_REGION

REGION Network 3: bit gotowości wspólny Z2
   // AUMA
   // MODACT MOK250
   RUNG wire#powerrail
      Contact( "AlwaysTRUE" )
      Contact( "isPowerOK" )
      wire#w1
      Contact( "isAUMA_Z_2" )
      Contact( "inputAumagotowośćZ_2" )
      wire#w2
      S_Coil( "isGotowość_Z_2" )
   END_RUNG
   RUNG wire#w1
      I_Contact( "isAUMA_Z_2" )
      I_Contact( "setAlarm_Moment_Z_2" )
   END_RUNG wire#w2
   // the same network as SCL:
   IF "AlwaysTRUE" AND "isPowerOK" AND (("isAUMA_Z_2" AND "inputAumagotowośćZ_2") OR (NOT "isAUMA_Z_2" AND NOT "setAlarm_Moment_Z_2")) THEN
       "isGotowość_Z_2" := TRUE;
   END_IF;
END_REGION

REGION Network 4: bit gotowości wspólny Z2
   // AUMA
   // MODACT MOK250
   RUNG wire#powerrail
      Contact( "AlwaysTRUE" )
      Contact( "isPowerOK" )
      wire#w1
      Contact( "isAUMA_Z_2" )
      I_Contact( "inputAumagotowośćZ_2" )
      wire#w2
      R_Coil( "isGotowość_Z_2" )
   END_RUNG
   RUNG wire#w1
      I_Contact( "isAUMA_Z_2" )
      Contact( "setAlarm_Moment_Z_2" )
   END_RUNG wire#w2
   RUNG wire#w1
      Contact( "Hbit_Alarm_Z2" )
      Coil( "CMD_Awaria_Z_2" )
   END_RUNG
   // the same network as SCL:
   #_w1 := "AlwaysTRUE" AND "isPowerOK";
   IF #_w1 AND (("isAUMA_Z_2" AND NOT "inputAumagotowośćZ_2") OR (NOT "isAUMA_Z_2" AND "setAlarm_Moment_Z_2")) THEN
       "isGotowość_Z_2" := FALSE;
   END_IF;
   "CMD_Awaria_Z_2" := #_w1 AND "Hbit_Alarm_Z2";
END_REGION

REGION Network 5: bit gotowości wspólny Z3
   // AUMA
   // MODACT MOK250
   RUNG wire#powerrail
      Contact( "AlwaysTRUE" )
      Contact( "isPowerOK" )
      wire#w1
      Contact( "isAUMA_Z_3" )
      Contact( "inputAumagotowośćZ_3" )
      wire#w2
      S_Coil( "isGotowość_Z_3" )
   END_RUNG
   RUNG wire#w1
      I_Contact( "isAUMA_Z_3" )
      I_Contact( "setAlarm_Moment_Z_3" )
   END_RUNG wire#w2
   // the same network as SCL:
   IF "AlwaysTRUE" AND "isPowerOK" AND (("isAUMA_Z_3" AND "inputAumagotowośćZ_3") OR (NOT "isAUMA_Z_3" AND NOT "setAlarm_Moment_Z_3")) THEN
       "isGotowość_Z_3" := TRUE;
   END_IF;
END_REGION

REGION Network 6: bit gotowości wspólny Z3
   // AUMA
   // MODACT MOK250
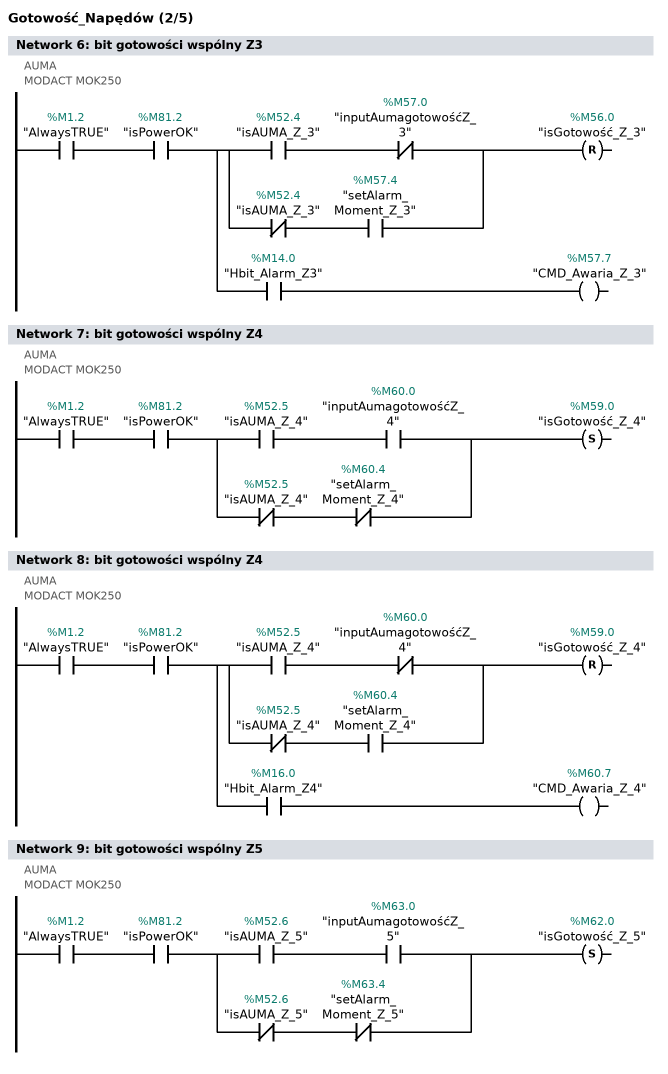
   RUNG wire#powerrail
      Contact( "AlwaysTRUE" )
      Contact( "isPowerOK" )
      wire#w1
      Contact( "isAUMA_Z_3" )
      I_Contact( "inputAumagotowośćZ_3" )
      wire#w2
      R_Coil( "isGotowość_Z_3" )
   END_RUNG
   RUNG wire#w1
      I_Contact( "isAUMA_Z_3" )
      Contact( "setAlarm_Moment_Z_3" )
   END_RUNG wire#w2
   RUNG wire#w1
      Contact( "Hbit_Alarm_Z3" )
      Coil( "CMD_Awaria_Z_3" )
   END_RUNG
   // the same network as SCL:
   #_w1 := "AlwaysTRUE" AND "isPowerOK";
   IF #_w1 AND (("isAUMA_Z_3" AND NOT "inputAumagotowośćZ_3") OR (NOT "isAUMA_Z_3" AND "setAlarm_Moment_Z_3")) THEN
       "isGotowość_Z_3" := FALSE;
   END_IF;
   "CMD_Awaria_Z_3" := #_w1 AND "Hbit_Alarm_Z3";
END_REGION

REGION Network 7: bit gotowości wspólny Z4
   // AUMA
   // MODACT MOK250
   RUNG wire#powerrail
      Contact( "AlwaysTRUE" )
      Contact( "isPowerOK" )
      wire#w1
      Contact( "isAUMA_Z_4" )
      Contact( "inputAumagotowośćZ_4" )
      wire#w2
      S_Coil( "isGotowość_Z_4" )
   END_RUNG
   RUNG wire#w1
      I_Contact( "isAUMA_Z_4" )
      I_Contact( "setAlarm_Moment_Z_4" )
   END_RUNG wire#w2
   // the same network as SCL:
   IF "AlwaysTRUE" AND "isPowerOK" AND (("isAUMA_Z_4" AND "inputAumagotowośćZ_4") OR (NOT "isAUMA_Z_4" AND NOT "setAlarm_Moment_Z_4")) THEN
       "isGotowość_Z_4" := TRUE;
   END_IF;
END_REGION

REGION Network 8: bit gotowości wspólny Z4
   // AUMA
   // MODACT MOK250
   RUNG wire#powerrail
      Contact( "AlwaysTRUE" )
      Contact( "isPowerOK" )
      wire#w1
      Contact( "isAUMA_Z_4" )
      I_Contact( "inputAumagotowośćZ_4" )
      wire#w2
      R_Coil( "isGotowość_Z_4" )
   END_RUNG
   RUNG wire#w1
      I_Contact( "isAUMA_Z_4" )
      Contact( "setAlarm_Moment_Z_4" )
   END_RUNG wire#w2
   RUNG wire#w1
      Contact( "Hbit_Alarm_Z4" )
      Coil( "CMD_Awaria_Z_4" )
   END_RUNG
   // the same network as SCL:
   #_w1 := "AlwaysTRUE" AND "isPowerOK";
   IF #_w1 AND (("isAUMA_Z_4" AND NOT "inputAumagotowośćZ_4") OR (NOT "isAUMA_Z_4" AND "setAlarm_Moment_Z_4")) THEN
       "isGotowość_Z_4" := FALSE;
   END_IF;
   "CMD_Awaria_Z_4" := #_w1 AND "Hbit_Alarm_Z4";
END_REGION

REGION Network 9: bit gotowości wspólny Z5
   // AUMA
   // MODACT MOK250
   RUNG wire#powerrail
      Contact( "AlwaysTRUE" )
      Contact( "isPowerOK" )
      wire#w1
      Contact( "isAUMA_Z_5" )
      Contact( "inputAumagotowośćZ_5" )
      wire#w2
      S_Coil( "isGotowość_Z_5" )
   END_RUNG
   RUNG wire#w1
      I_Contact( "isAUMA_Z_5" )
      I_Contact( "setAlarm_Moment_Z_5" )
   END_RUNG wire#w2
   // the same network as SCL:
   IF "AlwaysTRUE" AND "isPowerOK" AND (("isAUMA_Z_5" AND "inputAumagotowośćZ_5") OR (NOT "isAUMA_Z_5" AND NOT "setAlarm_Moment_Z_5")) THEN
       "isGotowość_Z_5" := TRUE;
   END_IF;
END_REGION

REGION Network 10: bit gotowości wspólny Z5
   // AUMA
   // MODACT MOK250
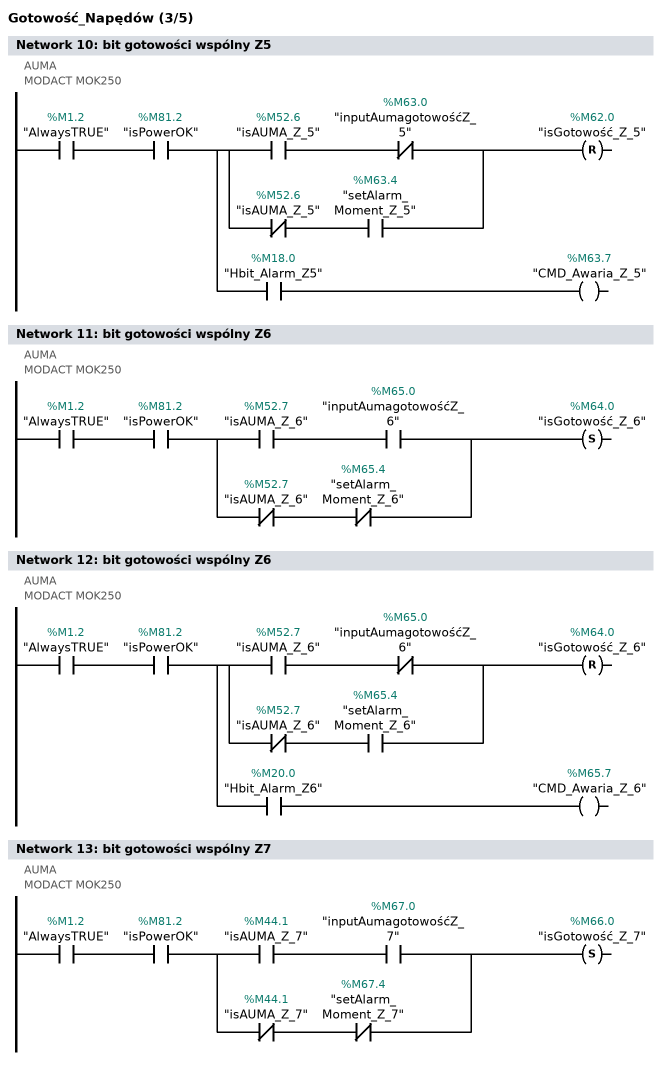
   RUNG wire#powerrail
      Contact( "AlwaysTRUE" )
      Contact( "isPowerOK" )
      wire#w1
      Contact( "isAUMA_Z_5" )
      I_Contact( "inputAumagotowośćZ_5" )
      wire#w2
      R_Coil( "isGotowość_Z_5" )
   END_RUNG
   RUNG wire#w1
      I_Contact( "isAUMA_Z_5" )
      Contact( "setAlarm_Moment_Z_5" )
   END_RUNG wire#w2
   RUNG wire#w1
      Contact( "Hbit_Alarm_Z5" )
      Coil( "CMD_Awaria_Z_5" )
   END_RUNG
   // the same network as SCL:
   #_w1 := "AlwaysTRUE" AND "isPowerOK";
   IF #_w1 AND (("isAUMA_Z_5" AND NOT "inputAumagotowośćZ_5") OR (NOT "isAUMA_Z_5" AND "setAlarm_Moment_Z_5")) THEN
       "isGotowość_Z_5" := FALSE;
   END_IF;
   "CMD_Awaria_Z_5" := #_w1 AND "Hbit_Alarm_Z5";
END_REGION

REGION Network 11: bit gotowości wspólny Z6
   // AUMA
   // MODACT MOK250
   RUNG wire#powerrail
      Contact( "AlwaysTRUE" )
      Contact( "isPowerOK" )
      wire#w1
      Contact( "isAUMA_Z_6" )
      Contact( "inputAumagotowośćZ_6" )
      wire#w2
      S_Coil( "isGotowość_Z_6" )
   END_RUNG
   RUNG wire#w1
      I_Contact( "isAUMA_Z_6" )
      I_Contact( "setAlarm_Moment_Z_6" )
   END_RUNG wire#w2
   // the same network as SCL:
   IF "AlwaysTRUE" AND "isPowerOK" AND (("isAUMA_Z_6" AND "inputAumagotowośćZ_6") OR (NOT "isAUMA_Z_6" AND NOT "setAlarm_Moment_Z_6")) THEN
       "isGotowość_Z_6" := TRUE;
   END_IF;
END_REGION

REGION Network 12: bit gotowości wspólny Z6
   // AUMA
   // MODACT MOK250
   RUNG wire#powerrail
      Contact( "AlwaysTRUE" )
      Contact( "isPowerOK" )
      wire#w1
      Contact( "isAUMA_Z_6" )
      I_Contact( "inputAumagotowośćZ_6" )
      wire#w2
      R_Coil( "isGotowość_Z_6" )
   END_RUNG
   RUNG wire#w1
      I_Contact( "isAUMA_Z_6" )
      Contact( "setAlarm_Moment_Z_6" )
   END_RUNG wire#w2
   RUNG wire#w1
      Contact( "Hbit_Alarm_Z6" )
      Coil( "CMD_Awaria_Z_6" )
   END_RUNG
   // the same network as SCL:
   #_w1 := "AlwaysTRUE" AND "isPowerOK";
   IF #_w1 AND (("isAUMA_Z_6" AND NOT "inputAumagotowośćZ_6") OR (NOT "isAUMA_Z_6" AND "setAlarm_Moment_Z_6")) THEN
       "isGotowość_Z_6" := FALSE;
   END_IF;
   "CMD_Awaria_Z_6" := #_w1 AND "Hbit_Alarm_Z6";
END_REGION

REGION Network 13: bit gotowości wspólny Z7
   // AUMA
   // MODACT MOK250
   RUNG wire#powerrail
      Contact( "AlwaysTRUE" )
      Contact( "isPowerOK" )
      wire#w1
      Contact( "isAUMA_Z_7" )
      Contact( "inputAumagotowośćZ_7" )
      wire#w2
      S_Coil( "isGotowość_Z_7" )
   END_RUNG
   RUNG wire#w1
      I_Contact( "isAUMA_Z_7" )
      I_Contact( "setAlarm_Moment_Z_7" )
   END_RUNG wire#w2
   // the same network as SCL:
   IF "AlwaysTRUE" AND "isPowerOK" AND (("isAUMA_Z_7" AND "inputAumagotowośćZ_7") OR (NOT "isAUMA_Z_7" AND NOT "setAlarm_Moment_Z_7")) THEN
       "isGotowość_Z_7" := TRUE;
   END_IF;
END_REGION

REGION Network 14: bit gotowości wspólny Z7
   // AUMA
   // MODACT MOK250
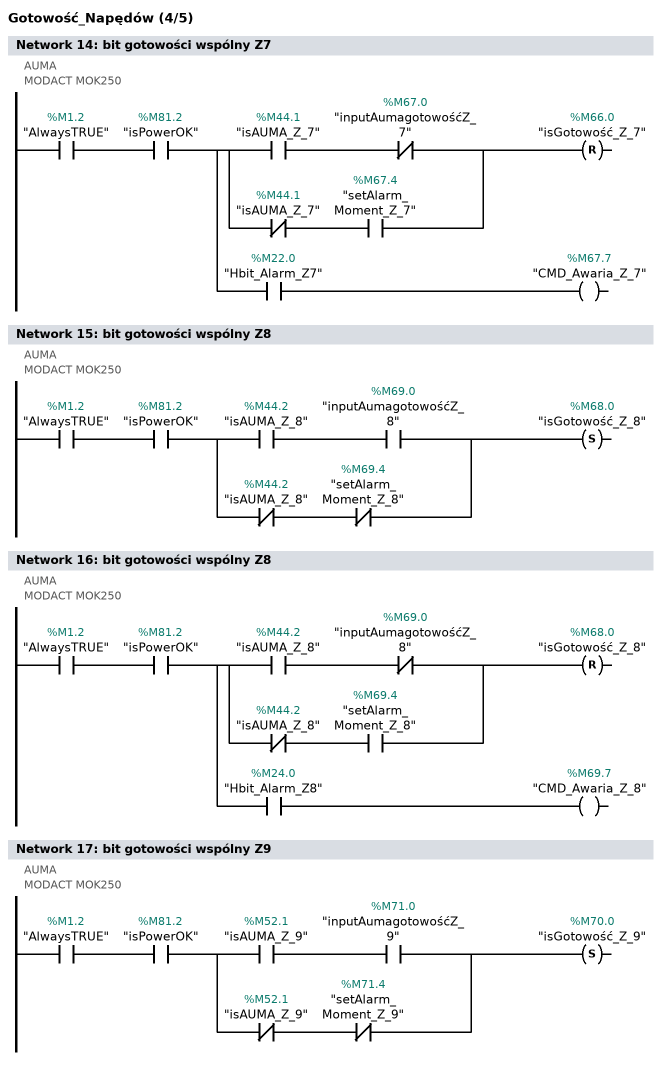
   RUNG wire#powerrail
      Contact( "AlwaysTRUE" )
      Contact( "isPowerOK" )
      wire#w1
      Contact( "isAUMA_Z_7" )
      I_Contact( "inputAumagotowośćZ_7" )
      wire#w2
      R_Coil( "isGotowość_Z_7" )
   END_RUNG
   RUNG wire#w1
      I_Contact( "isAUMA_Z_7" )
      Contact( "setAlarm_Moment_Z_7" )
   END_RUNG wire#w2
   RUNG wire#w1
      Contact( "Hbit_Alarm_Z7" )
      Coil( "CMD_Awaria_Z_7" )
   END_RUNG
   // the same network as SCL:
   #_w1 := "AlwaysTRUE" AND "isPowerOK";
   IF #_w1 AND (("isAUMA_Z_7" AND NOT "inputAumagotowośćZ_7") OR (NOT "isAUMA_Z_7" AND "setAlarm_Moment_Z_7")) THEN
       "isGotowość_Z_7" := FALSE;
   END_IF;
   "CMD_Awaria_Z_7" := #_w1 AND "Hbit_Alarm_Z7";
END_REGION

REGION Network 15: bit gotowości wspólny Z8
   // AUMA
   // MODACT MOK250
   RUNG wire#powerrail
      Contact( "AlwaysTRUE" )
      Contact( "isPowerOK" )
      wire#w1
      Contact( "isAUMA_Z_8" )
      Contact( "inputAumagotowośćZ_8" )
      wire#w2
      S_Coil( "isGotowość_Z_8" )
   END_RUNG
   RUNG wire#w1
      I_Contact( "isAUMA_Z_8" )
      I_Contact( "setAlarm_Moment_Z_8" )
   END_RUNG wire#w2
   // the same network as SCL:
   IF "AlwaysTRUE" AND "isPowerOK" AND (("isAUMA_Z_8" AND "inputAumagotowośćZ_8") OR (NOT "isAUMA_Z_8" AND NOT "setAlarm_Moment_Z_8")) THEN
       "isGotowość_Z_8" := TRUE;
   END_IF;
END_REGION

REGION Network 16: bit gotowości wspólny Z8
   // AUMA
   // MODACT MOK250
   RUNG wire#powerrail
      Contact( "AlwaysTRUE" )
      Contact( "isPowerOK" )
      wire#w1
      Contact( "isAUMA_Z_8" )
      I_Contact( "inputAumagotowośćZ_8" )
      wire#w2
      R_Coil( "isGotowość_Z_8" )
   END_RUNG
   RUNG wire#w1
      I_Contact( "isAUMA_Z_8" )
      Contact( "setAlarm_Moment_Z_8" )
   END_RUNG wire#w2
   RUNG wire#w1
      Contact( "Hbit_Alarm_Z8" )
      Coil( "CMD_Awaria_Z_8" )
   END_RUNG
   // the same network as SCL:
   #_w1 := "AlwaysTRUE" AND "isPowerOK";
   IF #_w1 AND (("isAUMA_Z_8" AND NOT "inputAumagotowośćZ_8") OR (NOT "isAUMA_Z_8" AND "setAlarm_Moment_Z_8")) THEN
       "isGotowość_Z_8" := FALSE;
   END_IF;
   "CMD_Awaria_Z_8" := #_w1 AND "Hbit_Alarm_Z8";
END_REGION

REGION Network 17: bit gotowości wspólny Z9
   // AUMA
   // MODACT MOK250
   RUNG wire#powerrail
      Contact( "AlwaysTRUE" )
      Contact( "isPowerOK" )
      wire#w1
      Contact( "isAUMA_Z_9" )
      Contact( "inputAumagotowośćZ_9" )
      wire#w2
      S_Coil( "isGotowość_Z_9" )
   END_RUNG
   RUNG wire#w1
      I_Contact( "isAUMA_Z_9" )
      I_Contact( "setAlarm_Moment_Z_9" )
   END_RUNG wire#w2
   // the same network as SCL:
   IF "AlwaysTRUE" AND "isPowerOK" AND (("isAUMA_Z_9" AND "inputAumagotowośćZ_9") OR (NOT "isAUMA_Z_9" AND NOT "setAlarm_Moment_Z_9")) THEN
       "isGotowość_Z_9" := TRUE;
   END_IF;
END_REGION

REGION Network 18: bit gotowości wspólny Z9
   // AUMA
   // MODACT MOK250
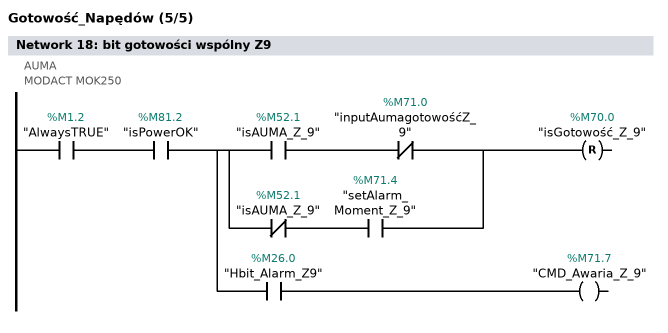
   RUNG wire#powerrail
      Contact( "AlwaysTRUE" )
      Contact( "isPowerOK" )
      wire#w1
      Contact( "isAUMA_Z_9" )
      I_Contact( "inputAumagotowośćZ_9" )
      wire#w2
      R_Coil( "isGotowość_Z_9" )
   END_RUNG
   RUNG wire#w1
      I_Contact( "isAUMA_Z_9" )
      Contact( "setAlarm_Moment_Z_9" )
   END_RUNG wire#w2
   RUNG wire#w1
      Contact( "Hbit_Alarm_Z9" )
      Coil( "CMD_Awaria_Z_9" )
   END_RUNG
   // the same network as SCL:
   #_w1 := "AlwaysTRUE" AND "isPowerOK";
   IF #_w1 AND (("isAUMA_Z_9" AND NOT "inputAumagotowośćZ_9") OR (NOT "isAUMA_Z_9" AND "setAlarm_Moment_Z_9")) THEN
       "isGotowość_Z_9" := FALSE;
   END_IF;
   "CMD_Awaria_Z_9" := #_w1 AND "Hbit_Alarm_Z9";
END_REGION
END_FUNCTION

FUNCTION_BLOCK "filtr _kalmana_2"
{ S7_Optimized_Access := 'TRUE' }
VERSION : 0.1

BEGIN
	IF "FirstScan" THEN //w pierwszym cyklu sterownika
	  FOR "I":= 0 TO 4 DO
	    "KALMAN_DB".kalman_K["I"] := 0.0;
	    "KALMAN_DB".kalman_R["I"] := 0.001;  //niepewność pomiaru
	    "KALMAN_DB".kalman_Q["I"] := 0.00001;  //niepewność procesu
	    "KALMAN_DB".kalman_P["I"] := 1.0;
	  END_FOR;        //parametry R i Q można dobrać osobno dla każdego kanału
	END_IF;           //zostaje wykonana inicjalizacja wszystkich 5 torów analogowych
	
	"R_TRIG_DB"(CLK:="Clock_10Hz",
	            Q=>"zbocze_dod_zegar"); //oczekiwanie na zbocze narastające
	
	IF "zbocze_dod_zegar" THEN  //ten fragment będzie wykonywany regularnie co 0.1s
	  
	  FOR "I":= 0 TO 4 DO
	  
	    "KALMAN_DB".wejscie_anal["I"] := PEEK_WORD(area:= 16#81, dbNumber:= 0, byteOffset:= (68 + (2 * "I")));
	    //sterownik odczytuje kolejno pięć wejść analogowych,
	    //kazde z nich zajmuje w pamięci jedno słowo począwszy od adresu %IW64
	    
	    //"KALMAN_DB".wejscie_anal["I"] := "KALMAN_DB".wejscie_anal["I"] AND 16#03FF;
	    //maskowanie wejść
	  
	    "KALMAN_DB".pomiar_napiecie["I"] := NORM_X(MIN:= 0, VALUE:= "KALMAN_DB".wejscie_anal["I"], MAX:= 27648);
	    //wartość zwracana przez n-bitowy przetwornik A\C zawiera się w przedziale od 0 do (2^n)-1
	  
	    "KALMAN_DB".pomiar_napiecie["I"] := "KALMAN_DB".pomiar_napiecie["I"] * 10.0;
	    //znormalizowana wartość zostaje pomnożona przez 10.0, aby tagi w tablicy "pomiar_napiecie"
	    //reprezentowały faktyczne napięcie na wejściu analogowym
	    //w przypadku zakresów wejściowych różnych od standardu można
	    //skorzystać z intruksji CASE i mnożyć wyjście przez różne skalary
	  
	    //FILTR KALMANA
	    "KALMAN_DB".kalman_P["I"] := "KALMAN_DB".kalman_P["I"] + "KALMAN_DB".kalman_Q["I"]; //predykcja
	  
	    "KALMAN_DB".kalman_K["I"] := "KALMAN_DB".kalman_P["I"] / ("KALMAN_DB".kalman_P["I"] + "KALMAN_DB".kalman_R["I"]); //korekcja
	    
	    "KALMAN_DB".kalman_napiecie["I"] := "KALMAN_DB".kalman_napiecie["I"] +
	                "KALMAN_DB".kalman_K["I"] * ("KALMAN_DB".pomiar_napiecie["I"] - "KALMAN_DB".kalman_napiecie["I"]);
	    
	    "KALMAN_DB".kalman_P["I"] := (1.0 - "KALMAN_DB".kalman_K["I"]) * "KALMAN_DB".kalman_P["I"];
	  
	    //wynik filtracji gotowy do użycia znajduje się w tablicy "KALMAN_DB".kalman_napiecie
	  
	  END_FOR;
	
	END_IF;
	
END_FUNCTION_BLOCK

FUNCTION "EX012_CheckErrorCounter" : Bool
TITLE = EX012_CheckErrorCounter
{ S7_Optimized_Access := 'TRUE' }
AUTHOR : RTEcmer
FAMILY : EX012
VERSION : 0.1
//Licznik błedów
   VAR_INPUT 
      CounterValue : USInt;
   END_VAR

   VAR_IN_OUT 
      PreviousCounterValue : USInt;
   END_VAR


BEGIN
	IF (#CounterValue <> #PreviousCounterValue) THEN
	    #EX012_CheckErrorCounter := TRUE;
	    #PreviousCounterValue := #CounterValue;
	ELSE
	    #EX012_CheckErrorCounter := FALSE;
	END_IF;
	    
	    
END_FUNCTION

FUNCTION "Error_Measurenment" : Void
TITLE = Handling error measurenment
{ S7_Optimized_Access := 'TRUE' }
AUTHOR : RTecmer
VERSION : 0.1
//The response to the loss of echo by the sonar and the result of the measurement of the difference will be taken.
   VAR_INPUT 
      Error_Echo1 : Bool;   // Signal loss echo sonar inflow
      Error_Echo2 : Bool;   // Signal loss echo sonar outlet
      Error_Level : Bool;   // Difference Level Error
   END_VAR

   VAR_OUTPUT 
      ErrorMeasurement : Bool;   // error relay
   END_VAR


BEGIN
	//If the echo error if the negative difference is set
	IF (#Error_Echo1 = TRUE OR #Error_Echo2 = TRUE ) THEN
	    #ErrorMeasurement := TRUE;
	ELSE
	    #ErrorMeasurement := FALSE;
	END_IF;
	    
	    
	
	
END_FUNCTION

FUNCTION "ERR_CompareSoftwareError" : Bool
{ S7_Optimized_Access := 'TRUE' }
VERSION : 0.1
   VAR_INPUT 
      Actual : DWord;
      Buffer : "stt_ERR_SoftwareError";
   END_VAR

   VAR_TEMP 
      tempCounter : USInt;
   END_VAR


BEGIN
	//searching difference
	#ERR_CompareSoftwareError := #Buffer.Status[#Buffer.Counter] <> #Actual;
	
	
END_FUNCTION

DATA_BLOCK "Startegia_sterowania_DB"   // DB72
AUTHOR : rtecmer
VERSION : 0.1
// stored: AutoNumber true, DBAccessibleFromOPCUA true, InstanceOfName Startegia_sterowania, InstanceOfType FB
"Startegia_sterowania"
BEGIN
END_DATA_BLOCK

DATA_BLOCK "godzinyPracy_DB-zb2"   // DB83
AUTHOR : RTecmer
FAMILY : XMHour
VERSION : 0.1
// stored: AutoNumber true, DBAccessibleFromOPCUA true, InstanceOfName godzinyPracy, InstanceOfType FB
"godzinyPracy"
BEGIN
END_DATA_BLOCK

DATA_BLOCK "godzinyPracy_DB_zb1"   // DB82
AUTHOR : RTecmer
FAMILY : XMHour
VERSION : 0.1
// stored: AutoNumber true, DBAccessibleFromOPCUA true, InstanceOfName godzinyPracy, InstanceOfType FB
"godzinyPracy"
BEGIN
END_DATA_BLOCK

DATA_BLOCK "godzinyPracy_DB_zb3"   // DB84
AUTHOR : RTecmer
FAMILY : XMHour
VERSION : 0.1
// stored: AutoNumber true, DBAccessibleFromOPCUA true, InstanceOfName godzinyPracy, InstanceOfType FB
"godzinyPracy"
BEGIN
END_DATA_BLOCK

DATA_BLOCK "godzinyPracy_DB_zb4"   // DB85
AUTHOR : RTecmer
FAMILY : XMHour
VERSION : 0.1
// stored: AutoNumber true, DBAccessibleFromOPCUA true, InstanceOfName godzinyPracy, InstanceOfType FB
"godzinyPracy"
BEGIN
END_DATA_BLOCK

DATA_BLOCK "FB220_TimeSyn_PLC_To_HMI_DB_1"   // DB78
VERSION : 0.1
// stored: AutoNumber true, DBAccessibleFromOPCUA true, InstanceOfName FB220_TimeSyn_PLC_To_HMI, InstanceOfType FB
"FB220_TimeSyn_PLC_To_HMI"
   // VAR_OUTPUT
   //    PLC_RD_LOC_T : DTL;
   //    PLC_RD_SYS_T : DTL;
   // END_VAR
   // VAR_IN_OUT
   //    AreaPointer_JobMailbox : Array[0..3] of Word;
   //    SetTime : Bool;
   //    SetDate : Bool;
   // END_VAR
   // VAR
   //    Func_RD_LOC_T : DTL;
   //    Ret_Val_RD_LOC_T : Int;
   //    BCD_Hour : Word;
   //    BCD_Minute : Word;
   //    BCD_Second : Word;
   //    BCD_Weekdday : Word;
   //    BCD_Day : Word;
   //    BCD_Month : Word;
   //    BCD32_Year : DWord;
   //    BCD16_Year : Word;
   //    STEP1 : Bool;
   //    STEP2 : Bool;
   //    STEP3 : Bool;
   //    STEP10 : Bool;
   //    STEP11 : Bool;
   //    STEP12 : Bool;
   //    Func_RD_SYS_T : DTL;
   //    Ret_Val_RD_SYS_T : Int;
   // END_VAR
BEGIN
END_DATA_BLOCK

DATA_BLOCK "AI_Scalowani_Położenia_Z10_DB"   // DB33
AUTHOR : rtecmer
VERSION : 0.1
// stored: AutoNumber true, DBAccessibleFromOPCUA true, InstanceOfName AI_Scalowani_Położenia_Z10, InstanceOfType FB
"AI_Scalowani_Położenia_Z10"
BEGIN
END_DATA_BLOCK

DATA_BLOCK "Byte Status Z1-Z10_DB"   // DB5
AUTHOR : rtecmer
VERSION : 0.1
// stored: AutoNumber true, DBAccessibleFromOPCUA true, InstanceOfName Byte Status Z1-Z10, InstanceOfType FB
"Byte Status Z1-Z10"
BEGIN
END_DATA_BLOCK

DATA_BLOCK "VLV02_POSITION_DB_Z10"   // DB26
AUTHOR : RTecmer
VERSION : 0.2
// stored: AutoNumber true, DBAccessibleFromOPCUA true, InstanceOfName VLV02_POSITION, InstanceOfType FB
"VLV02_POSITION"
BEGIN
END_DATA_BLOCK

DATA_BLOCK "WatchDog HMI_DB_1"   // DB40
AUTHOR : rtecmer
VERSION : 0.1
// stored: AutoNumber true, DBAccessibleFromOPCUA true, InstanceOfName WatchDog HMI, InstanceOfType FB
"WatchDog HMI"
BEGIN
END_DATA_BLOCK

DATA_BLOCK "generator_weekday_DB"   // DB49
AUTHOR : RTecmer
FAMILY : XMHour
VERSION : 0.1
// stored: AutoNumber true, DBAccessibleFromOPCUA true, InstanceOfName generator_weekday, InstanceOfType FB
"generator_weekday"
BEGIN
END_DATA_BLOCK

DATA_BLOCK "filtr _kalmana_1_DB"   // DB51
VERSION : 0.1
// stored: AutoNumber true, DBAccessibleFromOPCUA true, InstanceOfName filtr _kalmana_2, InstanceOfType FB
"filtr _kalmana_2"
BEGIN
END_DATA_BLOCK

DATA_BLOCK "VLV02_DB_Z1"   // DB13
AUTHOR : RTecmer
VERSION : 0.2
// stored: AutoNumber true, DBAccessibleFromOPCUA true, InstanceOfName VLV02, InstanceOfType FB
"VLV02"
BEGIN
END_DATA_BLOCK

DATA_BLOCK "VLV02_DB_Z2"   // DB14
AUTHOR : RTecmer
VERSION : 0.2
// stored: AutoNumber false, DBAccessibleFromOPCUA true, InstanceOfName VLV02, InstanceOfType FB
"VLV02"
BEGIN
END_DATA_BLOCK

DATA_BLOCK "VLV02_DB_Z4"   // DB16
AUTHOR : RTecmer
VERSION : 0.2
// stored: AutoNumber true, DBAccessibleFromOPCUA true, InstanceOfName VLV02, InstanceOfType FB
"VLV02"
BEGIN
END_DATA_BLOCK

DATA_BLOCK "VLV02_DB_Z5"   // DB17
AUTHOR : RTecmer
VERSION : 0.2
// stored: AutoNumber true, DBAccessibleFromOPCUA true, InstanceOfName VLV02, InstanceOfType FB
"VLV02"
BEGIN
END_DATA_BLOCK

DATA_BLOCK "VLV02_DB_Z6"   // DB18
AUTHOR : RTecmer
VERSION : 0.2
// stored: AutoNumber true, DBAccessibleFromOPCUA true, InstanceOfName VLV02, InstanceOfType FB
"VLV02"
BEGIN
END_DATA_BLOCK

DATA_BLOCK "VLV02_DB_Z7"   // DB19
AUTHOR : RTecmer
VERSION : 0.2
// stored: AutoNumber true, DBAccessibleFromOPCUA true, InstanceOfName VLV02, InstanceOfType FB
"VLV02"
BEGIN
END_DATA_BLOCK

DATA_BLOCK "VLV02_DB_Z8"   // DB20
AUTHOR : RTecmer
VERSION : 0.2
// stored: AutoNumber true, DBAccessibleFromOPCUA true, InstanceOfName VLV02, InstanceOfType FB
"VLV02"
BEGIN
END_DATA_BLOCK

DATA_BLOCK "VLV02_DB_Z9"   // DB21
AUTHOR : RTecmer
VERSION : 0.2
// stored: AutoNumber true, DBAccessibleFromOPCUA true, InstanceOfName VLV02, InstanceOfType FB
"VLV02"
BEGIN
END_DATA_BLOCK

DATA_BLOCK "VLV02_DB_z3"   // DB15
AUTHOR : RTecmer
VERSION : 0.2
// stored: AutoNumber false, DBAccessibleFromOPCUA true, InstanceOfName VLV02, InstanceOfType FB
"VLV02"
BEGIN
END_DATA_BLOCK

DATA_BLOCK "Alarm_magistrala_B5_DB"   // DB71
AUTHOR : rtecmer
VERSION : 0.1
// stored: AutoNumber true, DBAccessibleFromOPCUA true, InstanceOfName Alarm_magistrala_B5, InstanceOfType FB
"Alarm_magistrala_B5"
BEGIN
END_DATA_BLOCK

DATA_BLOCK "Client_ModbusTCP_read_DLT_DB"   // DB9
AUTHOR : rtecmer
VERSION : 0.1
// stored: AutoNumber true, DBAccessibleFromOPCUA true, InstanceOfName Client_ModbusTCP_read_DLT, InstanceOfType FB
"Client_ModbusTCP_read_DLT"
BEGIN
END_DATA_BLOCK

DATA_BLOCK "Client_ModbusTCP_read_control_DB"   // DB4
AUTHOR : rtecmer
VERSION : 0.1
// stored: AutoNumber true, DBAccessibleFromOPCUA true, InstanceOfName Client_ModbusTCP_read_control, InstanceOfType FB
"Client_ModbusTCP_read_control"
BEGIN
END_DATA_BLOCK

DATA_BLOCK "Client_ModbusTCP_sending_analogs_DB"   // DB11
AUTHOR : rtecmer
VERSION : 0.1
// stored: AutoNumber true, DBAccessibleFromOPCUA true, InstanceOfName Client_ModbusTCP_sending_analogs, InstanceOfType FB
"Client_ModbusTCP_sending_analogs"
BEGIN
END_DATA_BLOCK

DATA_BLOCK "Client_ModbusTCP_sending_parameters_DB"   // DB30
AUTHOR : rtecmer
VERSION : 0.1
// stored: AutoNumber true, DBAccessibleFromOPCUA true, InstanceOfName Client_ModbusTCP_sending_parameters, InstanceOfType FB
"Client_ModbusTCP_sending_parameters"
BEGIN
END_DATA_BLOCK

DATA_BLOCK "Client_ModbusTCP_sending_status_DB"   // DB27
AUTHOR : rtecmer
VERSION : 0.1
// stored: AutoNumber true, DBAccessibleFromOPCUA true, InstanceOfName Client_ModbusTCP_sending_status, InstanceOfType FB
"Client_ModbusTCP_sending_status"
BEGIN
END_DATA_BLOCK

DATA_BLOCK "EX012_ErrorHandling_DB"   // DB67
VERSION : 0.1
// stored: AutoNumber true, DBAccessibleFromOPCUA true, InstanceOfName EX012_ErrorHandling, InstanceOfType FB
"EX012_ErrorHandling"
BEGIN
END_DATA_BLOCK

DATA_BLOCK "IEC_Timer_Hist_SetHWork_P1_DB"   // DB47
{ S7_Optimized_Access := 'TRUE' }
// stored: AutoNumber true, DBAccessibleFromOPCUA true, InstanceOfName IEC_TIMER, OfSystemLibElement IEC_TIMER, OfSystemLibVersion 1.0
"IEC_TIMER"
   // VAR
   //    PT : Time;
   //    ET { ExternalWritable := 'False'} : Time;
   //    IN : Bool;
   //    Q { ExternalWritable := 'False'} : Bool;
   // END_VAR
BEGIN
END_DATA_BLOCK

DATA_BLOCK "IEC_Timer_Hist_SetHWork_P2_DB"   // DB74
{ S7_Optimized_Access := 'TRUE' }
// stored: AutoNumber true, DBAccessibleFromOPCUA true, InstanceOfName IEC_TIMER, OfSystemLibElement IEC_TIMER, OfSystemLibVersion 1.0
"IEC_TIMER"
   // VAR
   //    PT : Time;
   //    ET { ExternalWritable := 'False'} : Time;
   //    IN : Bool;
   //    Q { ExternalWritable := 'False'} : Bool;
   // END_VAR
BEGIN
END_DATA_BLOCK

DATA_BLOCK "IEC_Timer_My_1Hz_In_DB"   // DB88
{ S7_Optimized_Access := 'TRUE' }
// stored: AutoNumber true, DBAccessibleFromOPCUA true, InstanceOfName IEC_TIMER, OfSystemLibElement IEC_TIMER, OfSystemLibVersion 1.0
"IEC_TIMER"
   // VAR
   //    PT : Time;
   //    ET { ExternalWritable := 'False'} : Time;
   //    IN : Bool;
   //    Q { ExternalWritable := 'False'} : Bool;
   // END_VAR
BEGIN
END_DATA_BLOCK

DATA_BLOCK "IEC_Timer_My_1Hz_out_DB"   // DB89
{ S7_Optimized_Access := 'TRUE' }
// stored: AutoNumber true, DBAccessibleFromOPCUA true, InstanceOfName IEC_TIMER, OfSystemLibElement IEC_TIMER, OfSystemLibVersion 1.0
"IEC_TIMER"
   // VAR
   //    PT : Time;
   //    ET { ExternalWritable := 'False'} : Time;
   //    IN : Bool;
   //    Q { ExternalWritable := 'False'} : Bool;
   // END_VAR
BEGIN
END_DATA_BLOCK

DATA_BLOCK "IEC_Timer_PulseON_Z_DB"   // DB22
{ S7_Optimized_Access := 'TRUE' }
// stored: AutoNumber true, DBAccessibleFromOPCUA true, InstanceOfName IEC_TIMER, OfSystemLibElement IEC_TIMER, OfSystemLibVersion 1.0
"IEC_TIMER"
   // VAR
   //    PT : Time;
   //    ET { ExternalWritable := 'False'} : Time;
   //    IN : Bool;
   //    Q { ExternalWritable := 'False'} : Bool;
   // END_VAR
BEGIN
END_DATA_BLOCK

DATA_BLOCK "IEC_Timer_error_modbus_tcp_res_DB"   // DB42
{ S7_Optimized_Access := 'TRUE' }
// stored: AutoNumber false, DBAccessibleFromOPCUA true, InstanceOfName IEC_TIMER, OfSystemLibElement IEC_TIMER, OfSystemLibVersion 1.0
"IEC_TIMER"
   // VAR
   //    PT : Time;
   //    ET { ExternalWritable := 'False'} : Time;
   //    IN : Bool;
   //    Q { ExternalWritable := 'False'} : Bool;
   // END_VAR
BEGIN
END_DATA_BLOCK

DATA_BLOCK "IEC_Timer_loop_rtu_error_DB"   // DB65
{ S7_Optimized_Access := 'TRUE' }
// stored: AutoNumber true, DBAccessibleFromOPCUA true, InstanceOfName IEC_TIMER, OfSystemLibElement IEC_TIMER, OfSystemLibVersion 1.0
"IEC_TIMER"
   // VAR
   //    PT : Time;
   //    ET { ExternalWritable := 'False'} : Time;
   //    IN : Bool;
   //    Q { ExternalWritable := 'False'} : Bool;
   // END_VAR
BEGIN
END_DATA_BLOCK

DATA_BLOCK "IEC_Timer_onTCP_DB"   // DB46
{ S7_Optimized_Access := 'TRUE' }
// stored: AutoNumber true, DBAccessibleFromOPCUA true, InstanceOfName IEC_TIMER, OfSystemLibElement IEC_TIMER, OfSystemLibVersion 1.0
"IEC_TIMER"
   // VAR
   //    PT : Time;
   //    ET { ExternalWritable := 'False'} : Time;
   //    IN : Bool;
   //    Q { ExternalWritable := 'False'} : Bool;
   // END_VAR
BEGIN
END_DATA_BLOCK

DATA_BLOCK "IEC_Timer_pulseClose_Z_DB"   // DB25
{ S7_Optimized_Access := 'TRUE' }
// stored: AutoNumber true, DBAccessibleFromOPCUA true, InstanceOfName IEC_TIMER, OfSystemLibElement IEC_TIMER, OfSystemLibVersion 1.0
"IEC_TIMER"
   // VAR
   //    PT : Time;
   //    ET { ExternalWritable := 'False'} : Time;
   //    IN : Bool;
   //    Q { ExternalWritable := 'False'} : Bool;
   // END_VAR
BEGIN
END_DATA_BLOCK

DATA_BLOCK "IEC_Timer_pulseOff_Z_DB"   // DB24
{ S7_Optimized_Access := 'TRUE' }
// stored: AutoNumber true, DBAccessibleFromOPCUA true, InstanceOfName IEC_TIMER, OfSystemLibElement IEC_TIMER, OfSystemLibVersion 1.0
"IEC_TIMER"
   // VAR
   //    PT : Time;
   //    ET { ExternalWritable := 'False'} : Time;
   //    IN : Bool;
   //    Q { ExternalWritable := 'False'} : Bool;
   // END_VAR
BEGIN
END_DATA_BLOCK

DATA_BLOCK "IEC_Timer_pulseOpen_DB"   // DB23
{ S7_Optimized_Access := 'TRUE' }
// stored: AutoNumber true, DBAccessibleFromOPCUA true, InstanceOfName IEC_TIMER, OfSystemLibElement IEC_TIMER, OfSystemLibVersion 1.0
"IEC_TIMER"
   // VAR
   //    PT : Time;
   //    ET { ExternalWritable := 'False'} : Time;
   //    IN : Bool;
   //    Q { ExternalWritable := 'False'} : Bool;
   // END_VAR
BEGIN
END_DATA_BLOCK

DATA_BLOCK "IEC_Timer_reser_active3_DB"   // DB79
{ S7_Optimized_Access := 'TRUE' }
// stored: AutoNumber true, DBAccessibleFromOPCUA true, InstanceOfName IEC_TIMER, OfSystemLibElement IEC_TIMER, OfSystemLibVersion 1.0
"IEC_TIMER"
   // VAR
   //    PT : Time;
   //    ET { ExternalWritable := 'False'} : Time;
   //    IN : Bool;
   //    Q { ExternalWritable := 'False'} : Bool;
   // END_VAR
BEGIN
END_DATA_BLOCK

DATA_BLOCK "IEC_Timer_reset_activ2_DB"   // DB77
{ S7_Optimized_Access := 'TRUE' }
// stored: AutoNumber true, DBAccessibleFromOPCUA true, InstanceOfName IEC_TIMER, OfSystemLibElement IEC_TIMER, OfSystemLibVersion 1.0
"IEC_TIMER"
   // VAR
   //    PT : Time;
   //    ET { ExternalWritable := 'False'} : Time;
   //    IN : Bool;
   //    Q { ExternalWritable := 'False'} : Bool;
   // END_VAR
BEGIN
END_DATA_BLOCK

DATA_BLOCK "IEC_Timer_reset_active4_DB"   // DB80
{ S7_Optimized_Access := 'TRUE' }
// stored: AutoNumber true, DBAccessibleFromOPCUA true, InstanceOfName IEC_TIMER, OfSystemLibElement IEC_TIMER, OfSystemLibVersion 1.0
"IEC_TIMER"
   // VAR
   //    PT : Time;
   //    ET { ExternalWritable := 'False'} : Time;
   //    IN : Bool;
   //    Q { ExternalWritable := 'False'} : Bool;
   // END_VAR
BEGIN
END_DATA_BLOCK

DATA_BLOCK "IEC_Timer_reset_active_1_DB"   // DB73
{ S7_Optimized_Access := 'TRUE' }
// stored: AutoNumber true, DBAccessibleFromOPCUA true, InstanceOfName IEC_TIMER, OfSystemLibElement IEC_TIMER, OfSystemLibVersion 1.0
"IEC_TIMER"
   // VAR
   //    PT : Time;
   //    ET { ExternalWritable := 'False'} : Time;
   //    IN : Bool;
   //    Q { ExternalWritable := 'False'} : Bool;
   // END_VAR
BEGIN
END_DATA_BLOCK

DATA_BLOCK "IEC_Timer_set_HWork_P3_DB"   // DB75
{ S7_Optimized_Access := 'TRUE' }
// stored: AutoNumber true, DBAccessibleFromOPCUA true, InstanceOfName IEC_TIMER, OfSystemLibElement IEC_TIMER, OfSystemLibVersion 1.0
"IEC_TIMER"
   // VAR
   //    PT : Time;
   //    ET { ExternalWritable := 'False'} : Time;
   //    IN : Bool;
   //    Q { ExternalWritable := 'False'} : Bool;
   // END_VAR
BEGIN
END_DATA_BLOCK

DATA_BLOCK "IEC_Timer_set_HWork_P4_DB"   // DB76
{ S7_Optimized_Access := 'TRUE' }
// stored: AutoNumber true, DBAccessibleFromOPCUA true, InstanceOfName IEC_TIMER, OfSystemLibElement IEC_TIMER, OfSystemLibVersion 1.0
"IEC_TIMER"
   // VAR
   //    PT : Time;
   //    ET { ExternalWritable := 'False'} : Time;
   //    IN : Bool;
   //    Q { ExternalWritable := 'False'} : Bool;
   // END_VAR
BEGIN
END_DATA_BLOCK

DATA_BLOCK "MB_CLIENT_DB_receiving"   // DB3
// stored: AutoNumber true, DBAccessibleFromOPCUA true, InstanceOfName MB_CLIENT, OfSystemLibElement MB_CLIENT, OfSystemLibVersion 3.1
"MB_CLIENT"
   // VAR_INPUT
   //    REQ : Bool;
   //    DISCONNECT : Bool;
   //    CONNECT_ID : UInt;
   //    IP_OCTET_1 : USInt;
   //    IP_OCTET_2 : USInt;
   //    IP_OCTET_3 : USInt;
   //    IP_OCTET_4 : USInt;
   //    IP_PORT : UInt;
   //    MB_MODE : USInt;
   //    MB_DATA_ADDR : UDInt;
   //    MB_DATA_LEN : UInt;
   // END_VAR
   // VAR_OUTPUT
   //    DONE : Bool;
   //    BUSY : Bool;
   //    ERROR : Bool;
   //    STATUS : Word;
   // END_VAR
   // VAR_IN_OUT
   //    MB_DATA_PTR : Variant;
   // END_VAR
   // VAR
   //    TCON_SFB { S7_SetPoint := 'True'} : TCON;
   //    TDISCON_SFB { S7_SetPoint := 'True'} : TDISCON;
   //    TSEND_SFB { S7_SetPoint := 'True'} : TSEND;
   //    TRCV_SFB { S7_SetPoint := 'True'} : TRCV;
   //    TCON_PARAM { S7_SetPoint := 'True'} : TCON_Param;
   //    PF_FREQUENCY : Real;
   //    BLOCKED_PROC_TIMEOUT : Real;
   //    RCV_TIMEOUT : Real;
   //    CURRENT_TIME_VALUE : DWord;
   //    SAVED_TIME_VALUE : DWord;
   //    XMT_TIME : DWord;
   //    SAVED_CONNECT_ID : Word;
   //    SAVED_IP_PORT : Word;
   //    SAVED_MODE : Byte;
   //    SAVED_IP1 : Byte;
   //    SAVED_IP2 : Byte;
   //    SAVED_IP3 : Byte;
   //    SAVED_IP4 : Byte;
   //    SAVED_DATA_ADDR : DWord;
   //    SAVED_DATA_LEN : Word;
   //    MB_STATE : Word;
   //    COMM_SENT_COUNT : Word;
   //    BYTE_COUNT : Word;
   //    BYTE_COUNTB : Byte;
   //    SAVED_START_ADDR : Word;
   //    MB_TRANSACTION_ID : Word;
   //    MB_UNIT_ID : Word;
   //    RETRIES : Word;
   //    INIT_OK : Bool;
   //    ACTIVE : Bool;
   //    CONNECTED : Bool;
   //    SAVED_MA_REQ : Bool;
   // END_VAR
BEGIN
END_DATA_BLOCK

DATA_BLOCK "MB_CLIENT_Send_DB"   // DB2
// stored: AutoNumber true, DBAccessibleFromOPCUA true, InstanceOfName MB_CLIENT, OfSystemLibElement MB_CLIENT, OfSystemLibVersion 3.1
"MB_CLIENT"
   // VAR_INPUT
   //    REQ : Bool;
   //    DISCONNECT : Bool;
   //    CONNECT_ID : UInt;
   //    IP_OCTET_1 : USInt;
   //    IP_OCTET_2 : USInt;
   //    IP_OCTET_3 : USInt;
   //    IP_OCTET_4 : USInt;
   //    IP_PORT : UInt;
   //    MB_MODE : USInt;
   //    MB_DATA_ADDR : UDInt;
   //    MB_DATA_LEN : UInt;
   // END_VAR
   // VAR_OUTPUT
   //    DONE : Bool;
   //    BUSY : Bool;
   //    ERROR : Bool;
   //    STATUS : Word;
   // END_VAR
   // VAR_IN_OUT
   //    MB_DATA_PTR : Variant;
   // END_VAR
   // VAR
   //    TCON_SFB { S7_SetPoint := 'True'} : TCON;
   //    TDISCON_SFB { S7_SetPoint := 'True'} : TDISCON;
   //    TSEND_SFB { S7_SetPoint := 'True'} : TSEND;
   //    TRCV_SFB { S7_SetPoint := 'True'} : TRCV;
   //    TCON_PARAM { S7_SetPoint := 'True'} : TCON_Param;
   //    PF_FREQUENCY : Real;
   //    BLOCKED_PROC_TIMEOUT : Real;
   //    RCV_TIMEOUT : Real;
   //    CURRENT_TIME_VALUE : DWord;
   //    SAVED_TIME_VALUE : DWord;
   //    XMT_TIME : DWord;
   //    SAVED_CONNECT_ID : Word;
   //    SAVED_IP_PORT : Word;
   //    SAVED_MODE : Byte;
   //    SAVED_IP1 : Byte;
   //    SAVED_IP2 : Byte;
   //    SAVED_IP3 : Byte;
   //    SAVED_IP4 : Byte;
   //    SAVED_DATA_ADDR : DWord;
   //    SAVED_DATA_LEN : Word;
   //    MB_STATE : Word;
   //    COMM_SENT_COUNT : Word;
   //    BYTE_COUNT : Word;
   //    BYTE_COUNTB : Byte;
   //    SAVED_START_ADDR : Word;
   //    MB_TRANSACTION_ID : Word;
   //    MB_UNIT_ID : Word;
   //    RETRIES : Word;
   //    INIT_OK : Bool;
   //    ACTIVE : Bool;
   //    CONNECTED : Bool;
   //    SAVED_MA_REQ : Bool;
   // END_VAR
BEGIN
END_DATA_BLOCK

DATA_BLOCK "MB_CLIENT_receivingTime"   // DB41
// stored: AutoNumber true, DBAccessibleFromOPCUA true, InstanceOfName MB_CLIENT, OfSystemLibElement MB_CLIENT, OfSystemLibVersion 3.1
"MB_CLIENT"
   // VAR_INPUT
   //    REQ : Bool;
   //    DISCONNECT : Bool;
   //    CONNECT_ID : UInt;
   //    IP_OCTET_1 : USInt;
   //    IP_OCTET_2 : USInt;
   //    IP_OCTET_3 : USInt;
   //    IP_OCTET_4 : USInt;
   //    IP_PORT : UInt;
   //    MB_MODE : USInt;
   //    MB_DATA_ADDR : UDInt;
   //    MB_DATA_LEN : UInt;
   // END_VAR
   // VAR_OUTPUT
   //    DONE : Bool;
   //    BUSY : Bool;
   //    ERROR : Bool;
   //    STATUS : Word;
   // END_VAR
   // VAR_IN_OUT
   //    MB_DATA_PTR : Variant;
   // END_VAR
   // VAR
   //    TCON_SFB { S7_SetPoint := 'True'} : TCON;
   //    TDISCON_SFB { S7_SetPoint := 'True'} : TDISCON;
   //    TSEND_SFB { S7_SetPoint := 'True'} : TSEND;
   //    TRCV_SFB { S7_SetPoint := 'True'} : TRCV;
   //    TCON_PARAM { S7_SetPoint := 'True'} : TCON_Param;
   //    PF_FREQUENCY : Real;
   //    BLOCKED_PROC_TIMEOUT : Real;
   //    RCV_TIMEOUT : Real;
   //    CURRENT_TIME_VALUE : DWord;
   //    SAVED_TIME_VALUE : DWord;
   //    XMT_TIME : DWord;
   //    SAVED_CONNECT_ID : Word;
   //    SAVED_IP_PORT : Word;
   //    SAVED_MODE : Byte;
   //    SAVED_IP1 : Byte;
   //    SAVED_IP2 : Byte;
   //    SAVED_IP3 : Byte;
   //    SAVED_IP4 : Byte;
   //    SAVED_DATA_ADDR : DWord;
   //    SAVED_DATA_LEN : Word;
   //    MB_STATE : Word;
   //    COMM_SENT_COUNT : Word;
   //    BYTE_COUNT : Word;
   //    BYTE_COUNTB : Byte;
   //    SAVED_START_ADDR : Word;
   //    MB_TRANSACTION_ID : Word;
   //    MB_UNIT_ID : Word;
   //    RETRIES : Word;
   //    INIT_OK : Bool;
   //    ACTIVE : Bool;
   //    CONNECTED : Bool;
   //    SAVED_MA_REQ : Bool;
   // END_VAR
BEGIN
END_DATA_BLOCK

DATA_BLOCK "MB_COMM_LOAD_Master_DB"   // DB38
// stored: AutoNumber true, DBAccessibleFromOPCUA true, InstanceOfName MB_COMM_LOAD, OfSystemLibElement MB_COMM_LOAD, OfSystemLibVersion 2.1
"MB_COMM_LOAD"
   // VAR_INPUT
   //    REQ : Bool;
   //    PORT : PORT;
   //    BAUD : UDInt;
   //    PARITY : UInt;
   //    FLOW_CTRL : UInt;
   //    RTS_ON_DLY : UInt;
   //    RTS_OFF_DLY : UInt;
   //    RESP_TO : UInt;
   // END_VAR
   // VAR_OUTPUT
   //    DONE : Bool;
   //    ERROR : Bool;
   //    STATUS : Word;
   // END_VAR
   // VAR_IN_OUT
   //    MB_DB : MB_BASE;
   // END_VAR
   // VAR
   //    ICHAR_GAP : UInt;
   //    RETRIES : UInt;
   //    WRREC_STATUS : Word;
   //    RDREC_STATUS : Word;
   //    SFC_STATUS : Word;
   //    Port_CFG_SFB : Array[0..25] of Byte;
   //    Send_CFG_SFB : Array[0..16] of Byte;
   //    Rcv_CFG_SFB : Array[0..60] of Byte;
   //    STOP_BITS : USInt := 2;
   // END_VAR
BEGIN
END_DATA_BLOCK

DATA_BLOCK "MB_MASTER_DB"   // DB39
// stored: AutoNumber true, DBAccessibleFromOPCUA true, InstanceOfName MB_MASTER, OfSystemLibElement MB_MASTER, OfSystemLibVersion 2.2
"MB_MASTER"
   // // inherited from MB_BASE
   // VAR
   //    S_PORT : UInt;
   //    S_RESP_TO : UInt;
   //    S_ICHAR_GAP : UInt;
   //    S_RETRIES : UInt;
   // END_VAR
   // VAR_INPUT
   //    REQ : Bool;
   //    MB_ADDR : UInt;
   //    MODE : USInt;
   //    DATA_ADDR : UDInt;
   //    DATA_LEN : UInt;
   // END_VAR
   // VAR_OUTPUT
   //    DONE : Bool;
   //    BUSY : Bool;
   //    ERROR : Bool;
   //    STATUS : Word;
   // END_VAR
   // VAR_IN_OUT
   //    DATA_PTR : Variant;
   // END_VAR
   // VAR
   //    SEND_PTP_SFB : Array[0..11] of Byte;
   //    RCV_PTP_SFB : Array[0..11] of Byte;
   //    RCV_RST_SFB : Array[0..9] of Byte;
   //    PF_FREQUENCY : Real;
   //    BLOCKED_PROC_TIMEOUT : Real;
   //    CURRENT_TIME_VALUE : UDInt;
   //    SAVED_TIME_VALUE : UDInt;
   //    SAVED_SLAVE_ADDR : Word;
   //    SAVED_MODE : Word;
   //    SAVED_DATA_ADDR : DWord;
   //    SAVED_DATA_LEN : UInt;
   //    MB_STATE : UInt;
   //    COMM_SENT_COUNT : UInt;
   //    BYTE_COUNT : USInt;
   //    INIT_OK : Bool;
   //    ACTIVE : Bool;
   //    BROADCAST_FLAG : Bool;
   //    EXTENDED_ADDRESSING : Bool;
   //    SAVED_START_ADDR : UInt;
   //    TXBuf_Function_Offset : UDInt;
   //    TXBuf_Address_Offset : UDInt;
   //    TXBuf_Quantity_Offset : UDInt;
   // END_VAR
BEGIN
END_DATA_BLOCK

DATA_BLOCK "Nastawy_Parametrów_Sterownia_DB"   // DB69
AUTHOR : rtecmer
VERSION : 0.1
// stored: AutoNumber true, DBAccessibleFromOPCUA true, InstanceOfName Nastawy_Parametrów_Sterownia, InstanceOfType FB
"Nastawy_Parametrów_Sterownia"
BEGIN
END_DATA_BLOCK

DATA_BLOCK "R_TRIG_DB"   // DB48
// stored: AutoNumber true, DBAccessibleFromOPCUA true, InstanceOfName R_TRIG, OfSystemLibElement R_TRIG, OfSystemLibVersion 1.0
"R_TRIG"
   // VAR_INPUT
   //    CLK : Bool;
   // END_VAR
   // VAR_OUTPUT
   //    Q : Bool;
   // END_VAR
   // VAR
   //    Stat_Bit : Bool;
   // END_VAR
BEGIN
END_DATA_BLOCK

DATA_BLOCK "R_TRIG_DB_AUT_Z1"   // DB52
// stored: AutoNumber true, DBAccessibleFromOPCUA true, InstanceOfName R_TRIG, OfSystemLibElement R_TRIG, OfSystemLibVersion 1.0
"R_TRIG"
   // VAR_INPUT
   //    CLK : Bool;
   // END_VAR
   // VAR_OUTPUT
   //    Q : Bool;
   // END_VAR
   // VAR
   //    Stat_Bit : Bool;
   // END_VAR
BEGIN
END_DATA_BLOCK

DATA_BLOCK "R_TRIG_DB_AUT_Z10"   // DB64
// stored: AutoNumber true, DBAccessibleFromOPCUA true, InstanceOfName R_TRIG, OfSystemLibElement R_TRIG, OfSystemLibVersion 1.0
"R_TRIG"
   // VAR_INPUT
   //    CLK : Bool;
   // END_VAR
   // VAR_OUTPUT
   //    Q : Bool;
   // END_VAR
   // VAR
   //    Stat_Bit : Bool;
   // END_VAR
BEGIN
END_DATA_BLOCK

DATA_BLOCK "R_TRIG_DB_AUT_Z2"   // DB54
// stored: AutoNumber true, DBAccessibleFromOPCUA true, InstanceOfName R_TRIG, OfSystemLibElement R_TRIG, OfSystemLibVersion 1.0
"R_TRIG"
   // VAR_INPUT
   //    CLK : Bool;
   // END_VAR
   // VAR_OUTPUT
   //    Q : Bool;
   // END_VAR
   // VAR
   //    Stat_Bit : Bool;
   // END_VAR
BEGIN
END_DATA_BLOCK

DATA_BLOCK "R_TRIG_DB_AUT_Z3"   // DB55
// stored: AutoNumber true, DBAccessibleFromOPCUA true, InstanceOfName R_TRIG, OfSystemLibElement R_TRIG, OfSystemLibVersion 1.0
"R_TRIG"
   // VAR_INPUT
   //    CLK : Bool;
   // END_VAR
   // VAR_OUTPUT
   //    Q : Bool;
   // END_VAR
   // VAR
   //    Stat_Bit : Bool;
   // END_VAR
BEGIN
END_DATA_BLOCK

DATA_BLOCK "R_TRIG_DB_AUT_Z4"   // DB59
// stored: AutoNumber true, DBAccessibleFromOPCUA true, InstanceOfName R_TRIG, OfSystemLibElement R_TRIG, OfSystemLibVersion 1.0
"R_TRIG"
   // VAR_INPUT
   //    CLK : Bool;
   // END_VAR
   // VAR_OUTPUT
   //    Q : Bool;
   // END_VAR
   // VAR
   //    Stat_Bit : Bool;
   // END_VAR
BEGIN
END_DATA_BLOCK

DATA_BLOCK "R_TRIG_DB_AUT_Z5"   // DB56
// stored: AutoNumber true, DBAccessibleFromOPCUA true, InstanceOfName R_TRIG, OfSystemLibElement R_TRIG, OfSystemLibVersion 1.0
"R_TRIG"
   // VAR_INPUT
   //    CLK : Bool;
   // END_VAR
   // VAR_OUTPUT
   //    Q : Bool;
   // END_VAR
   // VAR
   //    Stat_Bit : Bool;
   // END_VAR
BEGIN
END_DATA_BLOCK

DATA_BLOCK "R_TRIG_DB_AUT_Z6"   // DB60
// stored: AutoNumber true, DBAccessibleFromOPCUA true, InstanceOfName R_TRIG, OfSystemLibElement R_TRIG, OfSystemLibVersion 1.0
"R_TRIG"
   // VAR_INPUT
   //    CLK : Bool;
   // END_VAR
   // VAR_OUTPUT
   //    Q : Bool;
   // END_VAR
   // VAR
   //    Stat_Bit : Bool;
   // END_VAR
BEGIN
END_DATA_BLOCK

DATA_BLOCK "R_TRIG_DB_AUT_Z7"   // DB61
// stored: AutoNumber true, DBAccessibleFromOPCUA true, InstanceOfName R_TRIG, OfSystemLibElement R_TRIG, OfSystemLibVersion 1.0
"R_TRIG"
   // VAR_INPUT
   //    CLK : Bool;
   // END_VAR
   // VAR_OUTPUT
   //    Q : Bool;
   // END_VAR
   // VAR
   //    Stat_Bit : Bool;
   // END_VAR
BEGIN
END_DATA_BLOCK

DATA_BLOCK "R_TRIG_DB_AUT_Z8"   // DB62
// stored: AutoNumber true, DBAccessibleFromOPCUA true, InstanceOfName R_TRIG, OfSystemLibElement R_TRIG, OfSystemLibVersion 1.0
"R_TRIG"
   // VAR_INPUT
   //    CLK : Bool;
   // END_VAR
   // VAR_OUTPUT
   //    Q : Bool;
   // END_VAR
   // VAR
   //    Stat_Bit : Bool;
   // END_VAR
BEGIN
END_DATA_BLOCK

DATA_BLOCK "R_TRIG_DB_AUT_Z9"   // DB63
// stored: AutoNumber true, DBAccessibleFromOPCUA true, InstanceOfName R_TRIG, OfSystemLibElement R_TRIG, OfSystemLibVersion 1.0
"R_TRIG"
   // VAR_INPUT
   //    CLK : Bool;
   // END_VAR
   // VAR_OUTPUT
   //    Q : Bool;
   // END_VAR
   // VAR
   //    Stat_Bit : Bool;
   // END_VAR
BEGIN
END_DATA_BLOCK

DATA_BLOCK "WatchDog HMI_DB"   // DB8
AUTHOR : rtecmer
VERSION : 0.1
// stored: AutoNumber true, DBAccessibleFromOPCUA true, InstanceOfName WatchDog HMI, InstanceOfType FB
"WatchDog HMI"
BEGIN
END_DATA_BLOCK

DATA_BLOCK "alarm_petli-rtu_tcp_DB"   // DB66
AUTHOR : rtecmer
VERSION : 0.1
// stored: AutoNumber true, DBAccessibleFromOPCUA true, InstanceOfName alarm_petli-rtu_tcp, InstanceOfType FB
"alarm_petli-rtu_tcp"
BEGIN
END_DATA_BLOCK

DATA_BLOCK "filtr _kalmana_2_DB"   // DB50
VERSION : 0.1
// stored: AutoNumber true, DBAccessibleFromOPCUA true, InstanceOfName filtr _kalmana_2, InstanceOfType FB
"filtr _kalmana_2"
BEGIN
END_DATA_BLOCK

DATA_BLOCK "operating_mode_select_aut-man_DB"   // DB53
AUTHOR : rtecmer
VERSION : 0.1
// stored: AutoNumber true, DBAccessibleFromOPCUA true, InstanceOfName operating_mode_select_aut-man, InstanceOfType FB
"operating_mode_select_aut-man"
BEGIN
END_DATA_BLOCK

DATA_BLOCK "IEC_Timer_reserAlarmNiskie_cisnienie_DB"   // DB68
{ S7_Optimized_Access := 'TRUE' }
// stored: AutoNumber true, DBAccessibleFromOPCUA true, InstanceOfName IEC_TIMER, OfSystemLibElement IEC_TIMER, OfSystemLibVersion 1.0
"IEC_TIMER"
   // VAR
   //    PT : Time;
   //    ET { ExternalWritable := 'False'} : Time;
   //    IN : Bool;
   //    Q { ExternalWritable := 'False'} : Bool;
   // END_VAR
BEGIN
END_DATA_BLOCK

DATA_BLOCK "IEC_Timer_setAlarmNiskie_ciśnienie_DB"   // DB70
{ S7_Optimized_Access := 'TRUE' }
// stored: AutoNumber true, DBAccessibleFromOPCUA true, InstanceOfName IEC_TIMER, OfSystemLibElement IEC_TIMER, OfSystemLibVersion 1.0
"IEC_TIMER"
   // VAR
   //    PT : Time;
   //    ET { ExternalWritable := 'False'} : Time;
   //    IN : Bool;
   //    Q { ExternalWritable := 'False'} : Bool;
   // END_VAR
BEGIN
END_DATA_BLOCK

DATA_BLOCK "EX012_IDB8_ErrorHandling"   // DB104
VERSION : 0.1
// stored: AutoNumber false, DBAccessibleFromOPCUA true, InstanceOfName EX012_ErrorHandling, InstanceOfType FB
"EX012_ErrorHandling"
BEGIN
END_DATA_BLOCK
